REGION Network 15: Oscillator Screen Buttons
   // Set Buttons on based on operations of oscillator
   // Start Button on if Oscillating - State between 200-299
   // Hold Button on if Holding or Bumping - State between 100-199
   // Stop Button on if System Enabled but not Oscillating or Holding/Bumping awaiting Cmd- State 1
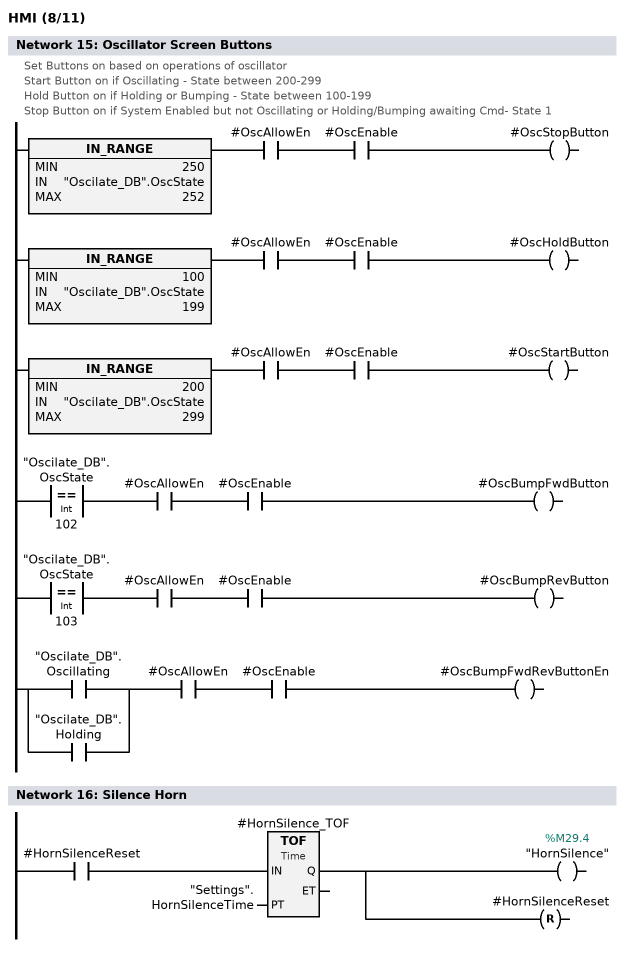
   RUNG wire#powerrail
      { S7_Templates := "SrcType := Int" } InRange(min := 250, in := "Oscilate_DB".OscState, max := 252)
      Contact( #OscAllowEn )
      Contact( #OscEnable )
      Coil( #OscStopButton )
   END_RUNG
   RUNG wire#powerrail
      { S7_Templates := "SrcType := Int" } InRange(min := 100, in := "Oscilate_DB".OscState, max := 199)
      Contact( #OscAllowEn )
      Contact( #OscEnable )
      Coil( #OscHoldButton )
   END_RUNG
   RUNG wire#powerrail
      { S7_Templates := "SrcType := Int" } InRange(min := 200, in := "Oscilate_DB".OscState, max := 299)
      Contact( #OscAllowEn )
      Contact( #OscEnable )
      Coil( #OscStartButton )
   END_RUNG
   RUNG wire#powerrail
      { S7_Templates := "SrcType := Int" } EQ_Contact(in1 := "Oscilate_DB".OscState, in2 := 102)
      Contact( #OscAllowEn )
      Contact( #OscEnable )
      Coil( #OscBumpFwdButton )
   END_RUNG
   RUNG wire#powerrail
      { S7_Templates := "SrcType := Int" } EQ_Contact(in1 := "Oscilate_DB".OscState, in2 := 103)
      Contact( #OscAllowEn )
      Contact( #OscEnable )
      Coil( #OscBumpRevButton )
   END_RUNG
   RUNG wire#powerrail
      Contact( "Oscilate_DB".Oscillating )
      wire#w1
      Contact( #OscAllowEn )
      Contact( #OscEnable )
      Coil( #OscBumpFwdRevButtonEn )
   END_RUNG
   RUNG wire#powerrail
      Contact( "Oscilate_DB".Holding )
   END_RUNG wire#w1
   // the same network as SCL:
   #OscStopButton := (250 <= "Oscilate_DB".OscState) AND ("Oscilate_DB".OscState <= 252) AND #OscAllowEn AND #OscEnable;
   #OscHoldButton := (100 <= "Oscilate_DB".OscState) AND ("Oscilate_DB".OscState <= 199) AND #OscAllowEn AND #OscEnable;
   #OscStartButton := (200 <= "Oscilate_DB".OscState) AND ("Oscilate_DB".OscState <= 299) AND #OscAllowEn AND #OscEnable;
   #OscBumpFwdButton := ("Oscilate_DB".OscState = 102) AND #OscAllowEn AND #OscEnable;
   #OscBumpRevButton := ("Oscilate_DB".OscState = 103) AND #OscAllowEn AND #OscEnable;
   #OscBumpFwdRevButtonEn := ("Oscilate_DB".Oscillating OR "Oscilate_DB".Holding) AND #OscAllowEn AND #OscEnable;
END_REGION

REGION Network 16: Silence Horn
   RUNG wire#powerrail
      Contact( #HornSilenceReset )
      { S7_Templates := "time_type := Time" } #HornSilence_TOF.TOF(pt := "Settings".HornSilenceTime, et =>)
      wire#w1
      Coil( "HornSilence" )
   END_RUNG
   RUNG wire#w1
      R_Coil( #HornSilenceReset )
   END_RUNG
   // the same network as SCL:
   #HornSilence_TOF(IN := #HornSilenceReset, PT := "Settings".HornSilenceTime);   // TOF
   "HornSilence" := #HornSilence_TOF.Q;
   IF #HornSilence_TOF.Q THEN #HornSilenceReset := FALSE; END_IF;
END_REGION

REGION Network 17: Assign Alarms to Alarms1 Int
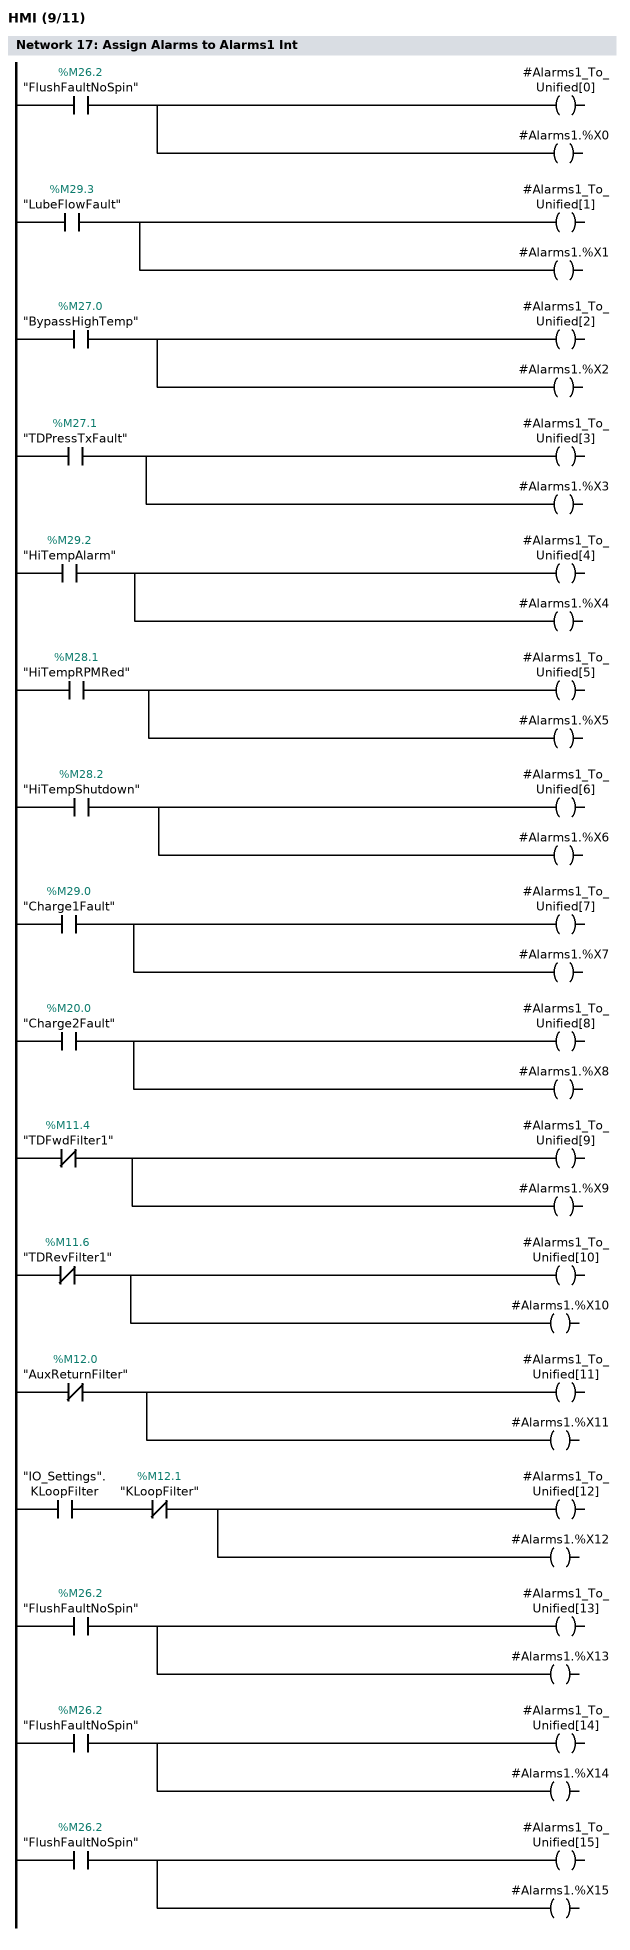
   RUNG wire#powerrail
      Contact( "FlushFaultNoSpin" )
      wire#w1
      Coil( #Alarms1_To_Unified[0] )
   END_RUNG
   RUNG wire#w1
      Coil( #Alarms1.%X0 )
   END_RUNG
   RUNG wire#powerrail
      Contact( "LubeFlowFault" )
      wire#w2
      Coil( #Alarms1_To_Unified[1] )
   END_RUNG
   RUNG wire#w2
      Coil( #Alarms1.%X1 )
   END_RUNG
   RUNG wire#powerrail
      Contact( "BypassHighTemp" )
      wire#w3
      Coil( #Alarms1_To_Unified[2] )
   END_RUNG
   RUNG wire#w3
      Coil( #Alarms1.%X2 )
   END_RUNG
   RUNG wire#powerrail
      Contact( "TDPressTxFault" )
      wire#w4
      Coil( #Alarms1_To_Unified[3] )
   END_RUNG
   RUNG wire#w4
      Coil( #Alarms1.%X3 )
   END_RUNG
   RUNG wire#powerrail
      Contact( "HiTempAlarm" )
      wire#w5
      Coil( #Alarms1_To_Unified[4] )
   END_RUNG
   RUNG wire#w5
      Coil( #Alarms1.%X4 )
   END_RUNG
   RUNG wire#powerrail
      Contact( "HiTempRPMRed" )
      wire#w6
      Coil( #Alarms1_To_Unified[5] )
   END_RUNG
   RUNG wire#w6
      Coil( #Alarms1.%X5 )
   END_RUNG
   RUNG wire#powerrail
      Contact( "HiTempShutdown" )
      wire#w7
      Coil( #Alarms1_To_Unified[6] )
   END_RUNG
   RUNG wire#w7
      Coil( #Alarms1.%X6 )
   END_RUNG
   RUNG wire#powerrail
      Contact( "Charge1Fault" )
      wire#w8
      Coil( #Alarms1_To_Unified[7] )
   END_RUNG
   RUNG wire#w8
      Coil( #Alarms1.%X7 )
   END_RUNG
   RUNG wire#powerrail
      Contact( "Charge2Fault" )
      wire#w9
      Coil( #Alarms1_To_Unified[8] )
   END_RUNG
   RUNG wire#w9
      Coil( #Alarms1.%X8 )
   END_RUNG
   RUNG wire#powerrail
      I_Contact( "TDFwdFilter1" )
      wire#w10
      Coil( #Alarms1_To_Unified[9] )
   END_RUNG
   RUNG wire#w10
      Coil( #Alarms1.%X9 )
   END_RUNG
   RUNG wire#powerrail
      I_Contact( "TDRevFilter1" )
      wire#w11
      Coil( #Alarms1_To_Unified[10] )
   END_RUNG
   RUNG wire#w11
      Coil( #Alarms1.%X10 )
   END_RUNG
   RUNG wire#powerrail
      I_Contact( "AuxReturnFilter" )
      wire#w12
      Coil( #Alarms1_To_Unified[11] )
   END_RUNG
   RUNG wire#w12
      Coil( #Alarms1.%X11 )
   END_RUNG
   RUNG wire#powerrail
      Contact( "IO_Settings".KLoopFilter )
      I_Contact( "KLoopFilter" )
      wire#w13
      Coil( #Alarms1_To_Unified[12] )
   END_RUNG
   RUNG wire#w13
      Coil( #Alarms1.%X12 )
   END_RUNG
   RUNG wire#powerrail
      Contact( "FlushFaultNoSpin" )
      wire#w14
      Coil( #Alarms1_To_Unified[13] )
   END_RUNG
   RUNG wire#w14
      Coil( #Alarms1.%X13 )
   END_RUNG
   RUNG wire#powerrail
      Contact( "FlushFaultNoSpin" )
      wire#w15
      Coil( #Alarms1_To_Unified[14] )
   END_RUNG
   RUNG wire#w15
      Coil( #Alarms1.%X14 )
   END_RUNG
   RUNG wire#powerrail
      Contact( "FlushFaultNoSpin" )
      wire#w16
      Coil( #Alarms1_To_Unified[15] )
   END_RUNG
   RUNG wire#w16
      Coil( #Alarms1.%X15 )
   END_RUNG
   // the same network as SCL:
   #Alarms1_To_Unified[0] := "FlushFaultNoSpin";
   #Alarms1.%X0 := "FlushFaultNoSpin";
   #Alarms1_To_Unified[1] := "LubeFlowFault";
   #Alarms1.%X1 := "LubeFlowFault";
   #Alarms1_To_Unified[2] := "BypassHighTemp";
   #Alarms1.%X2 := "BypassHighTemp";
   #Alarms1_To_Unified[3] := "TDPressTxFault";
   #Alarms1.%X3 := "TDPressTxFault";
   #Alarms1_To_Unified[4] := "HiTempAlarm";
   #Alarms1.%X4 := "HiTempAlarm";
   #Alarms1_To_Unified[5] := "HiTempRPMRed";
   #Alarms1.%X5 := "HiTempRPMRed";
   #Alarms1_To_Unified[6] := "HiTempShutdown";
   #Alarms1.%X6 := "HiTempShutdown";
   #Alarms1_To_Unified[7] := "Charge1Fault";
   #Alarms1.%X7 := "Charge1Fault";
   #Alarms1_To_Unified[8] := "Charge2Fault";
   #Alarms1.%X8 := "Charge2Fault";
   #Alarms1_To_Unified[9] := NOT "TDFwdFilter1";
   #Alarms1.%X9 := NOT "TDFwdFilter1";
   #Alarms1_To_Unified[10] := NOT "TDRevFilter1";
   #Alarms1.%X10 := NOT "TDRevFilter1";
   #Alarms1_To_Unified[11] := NOT "AuxReturnFilter";
   #Alarms1.%X11 := NOT "AuxReturnFilter";
   #Alarms1_To_Unified[12] := "IO_Settings".KLoopFilter AND NOT "KLoopFilter";
   #Alarms1.%X12 := "IO_Settings".KLoopFilter AND NOT "KLoopFilter";
   #Alarms1_To_Unified[13] := "FlushFaultNoSpin";
   #Alarms1.%X13 := "FlushFaultNoSpin";
   #Alarms1_To_Unified[14] := "FlushFaultNoSpin";
   #Alarms1.%X14 := "FlushFaultNoSpin";
   #Alarms1_To_Unified[15] := "FlushFaultNoSpin";
   #Alarms1.%X15 := "FlushFaultNoSpin";
END_REGION

REGION Network 18: Assign Alarms to Alarms2 Int
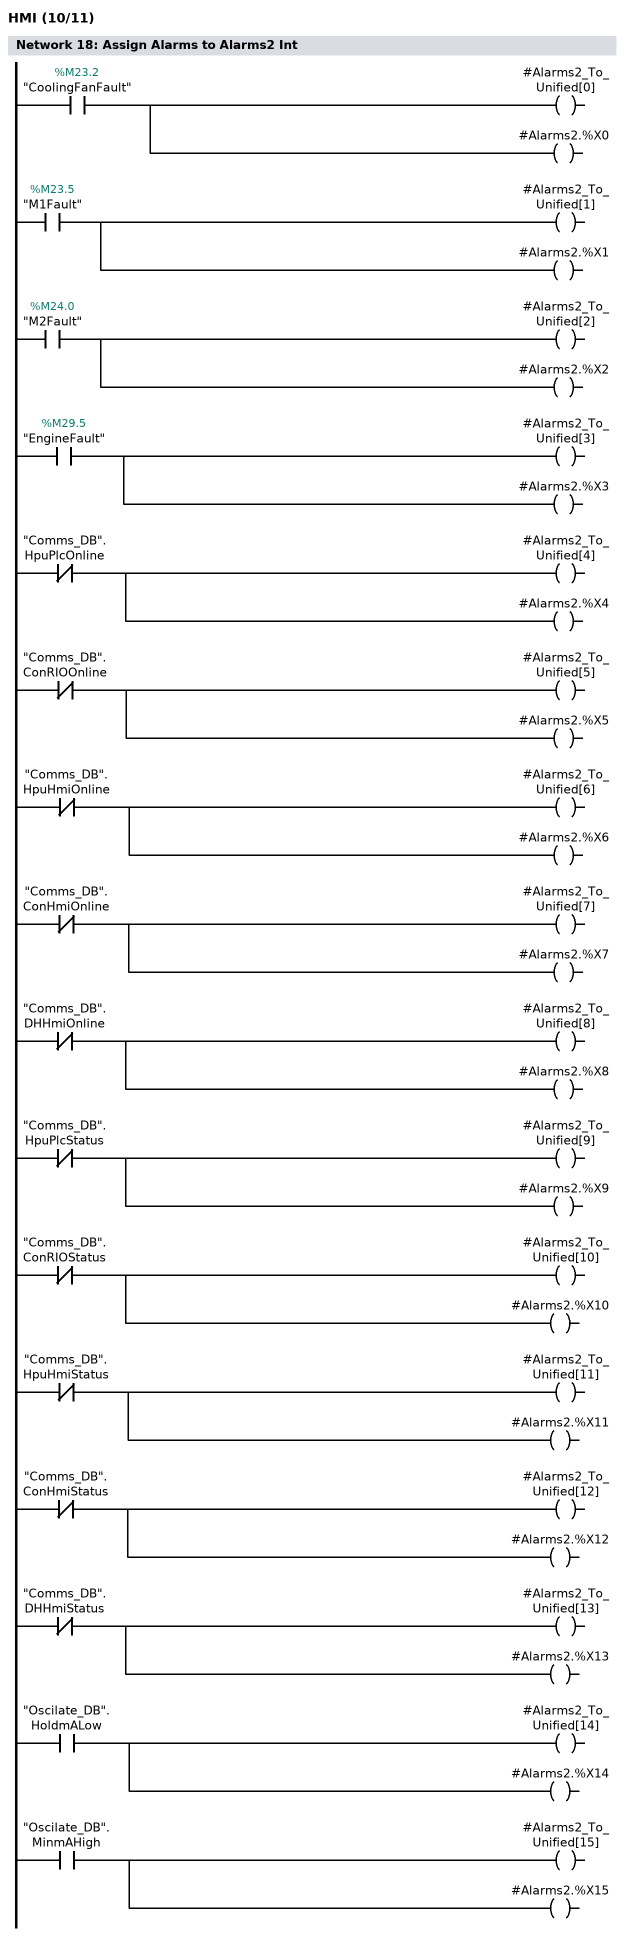
   RUNG wire#powerrail
      Contact( "CoolingFanFault" )
      wire#w1
      Coil( #Alarms2_To_Unified[0] )
   END_RUNG
   RUNG wire#w1
      Coil( #Alarms2.%X0 )
   END_RUNG
   RUNG wire#powerrail
      Contact( "M1Fault" )
      wire#w2
      Coil( #Alarms2_To_Unified[1] )
   END_RUNG
   RUNG wire#w2
      Coil( #Alarms2.%X1 )
   END_RUNG
   RUNG wire#powerrail
      Contact( "M2Fault" )
      wire#w3
      Coil( #Alarms2_To_Unified[2] )
   END_RUNG
   RUNG wire#w3
      Coil( #Alarms2.%X2 )
   END_RUNG
   RUNG wire#powerrail
      Contact( "EngineFault" )
      wire#w4
      Coil( #Alarms2_To_Unified[3] )
   END_RUNG
   RUNG wire#w4
      Coil( #Alarms2.%X3 )
   END_RUNG
   RUNG wire#powerrail
      I_Contact( "Comms_DB".HpuPlcOnline )
      wire#w5
      Coil( #Alarms2_To_Unified[4] )
   END_RUNG
   RUNG wire#w5
      Coil( #Alarms2.%X4 )
   END_RUNG
   RUNG wire#powerrail
      I_Contact( "Comms_DB".ConRIOOnline )
      wire#w6
      Coil( #Alarms2_To_Unified[5] )
   END_RUNG
   RUNG wire#w6
      Coil( #Alarms2.%X5 )
   END_RUNG
   RUNG wire#powerrail
      I_Contact( "Comms_DB".HpuHmiOnline )
      wire#w7
      Coil( #Alarms2_To_Unified[6] )
   END_RUNG
   RUNG wire#w7
      Coil( #Alarms2.%X6 )
   END_RUNG
   RUNG wire#powerrail
      I_Contact( "Comms_DB".ConHmiOnline )
      wire#w8
      Coil( #Alarms2_To_Unified[7] )
   END_RUNG
   RUNG wire#w8
      Coil( #Alarms2.%X7 )
   END_RUNG
   RUNG wire#powerrail
      I_Contact( "Comms_DB".DHHmiOnline )
      wire#w9
      Coil( #Alarms2_To_Unified[8] )
   END_RUNG
   RUNG wire#w9
      Coil( #Alarms2.%X8 )
   END_RUNG
   RUNG wire#powerrail
      I_Contact( "Comms_DB".HpuPlcStatus )
      wire#w10
      Coil( #Alarms2_To_Unified[9] )
   END_RUNG
   RUNG wire#w10
      Coil( #Alarms2.%X9 )
   END_RUNG
   RUNG wire#powerrail
      I_Contact( "Comms_DB".ConRIOStatus )
      wire#w11
      Coil( #Alarms2_To_Unified[10] )
   END_RUNG
   RUNG wire#w11
      Coil( #Alarms2.%X10 )
   END_RUNG
   RUNG wire#powerrail
      I_Contact( "Comms_DB".HpuHmiStatus )
      wire#w12
      Coil( #Alarms2_To_Unified[11] )
   END_RUNG
   RUNG wire#w12
      Coil( #Alarms2.%X11 )
   END_RUNG
   RUNG wire#powerrail
      I_Contact( "Comms_DB".ConHmiStatus )
      wire#w13
      Coil( #Alarms2_To_Unified[12] )
   END_RUNG
   RUNG wire#w13
      Coil( #Alarms2.%X12 )
   END_RUNG
   RUNG wire#powerrail
      I_Contact( "Comms_DB".DHHmiStatus )
      wire#w14
      Coil( #Alarms2_To_Unified[13] )
   END_RUNG
   RUNG wire#w14
      Coil( #Alarms2.%X13 )
   END_RUNG
   RUNG wire#powerrail
      Contact( "Oscilate_DB".HoldmALow )
      wire#w15
      Coil( #Alarms2_To_Unified[14] )
   END_RUNG
   RUNG wire#w15
      Coil( #Alarms2.%X14 )
   END_RUNG
   RUNG wire#powerrail
      Contact( "Oscilate_DB".MinmAHigh )
      wire#w16
      Coil( #Alarms2_To_Unified[15] )
   END_RUNG
   RUNG wire#w16
      Coil( #Alarms2.%X15 )
   END_RUNG
   // the same network as SCL:
   #Alarms2_To_Unified[0] := "CoolingFanFault";
   #Alarms2.%X0 := "CoolingFanFault";
   #Alarms2_To_Unified[1] := "M1Fault";
   #Alarms2.%X1 := "M1Fault";
   #Alarms2_To_Unified[2] := "M2Fault";
   #Alarms2.%X2 := "M2Fault";
   #Alarms2_To_Unified[3] := "EngineFault";
   #Alarms2.%X3 := "EngineFault";
   #Alarms2_To_Unified[4] := NOT "Comms_DB".HpuPlcOnline;
   #Alarms2.%X4 := NOT "Comms_DB".HpuPlcOnline;
   #Alarms2_To_Unified[5] := NOT "Comms_DB".ConRIOOnline;
   #Alarms2.%X5 := NOT "Comms_DB".ConRIOOnline;
   #Alarms2_To_Unified[6] := NOT "Comms_DB".HpuHmiOnline;
   #Alarms2.%X6 := NOT "Comms_DB".HpuHmiOnline;
   #Alarms2_To_Unified[7] := NOT "Comms_DB".ConHmiOnline;
   #Alarms2.%X7 := NOT "Comms_DB".ConHmiOnline;
   #Alarms2_To_Unified[8] := NOT "Comms_DB".DHHmiOnline;
   #Alarms2.%X8 := NOT "Comms_DB".DHHmiOnline;
   #Alarms2_To_Unified[9] := NOT "Comms_DB".HpuPlcStatus;
   #Alarms2.%X9 := NOT "Comms_DB".HpuPlcStatus;
   #Alarms2_To_Unified[10] := NOT "Comms_DB".ConRIOStatus;
   #Alarms2.%X10 := NOT "Comms_DB".ConRIOStatus;
   #Alarms2_To_Unified[11] := NOT "Comms_DB".HpuHmiStatus;
   #Alarms2.%X11 := NOT "Comms_DB".HpuHmiStatus;
   #Alarms2_To_Unified[12] := NOT "Comms_DB".ConHmiStatus;
   #Alarms2.%X12 := NOT "Comms_DB".ConHmiStatus;
   #Alarms2_To_Unified[13] := NOT "Comms_DB".DHHmiStatus;
   #Alarms2.%X13 := NOT "Comms_DB".DHHmiStatus;
   #Alarms2_To_Unified[14] := "Oscilate_DB".HoldmALow;
   #Alarms2.%X14 := "Oscilate_DB".HoldmALow;
   #Alarms2_To_Unified[15] := "Oscilate_DB".MinmAHigh;
   #Alarms2.%X15 := "Oscilate_DB".MinmAHigh;
END_REGION

REGION Network 19: Assign Warnings to Warnings Int
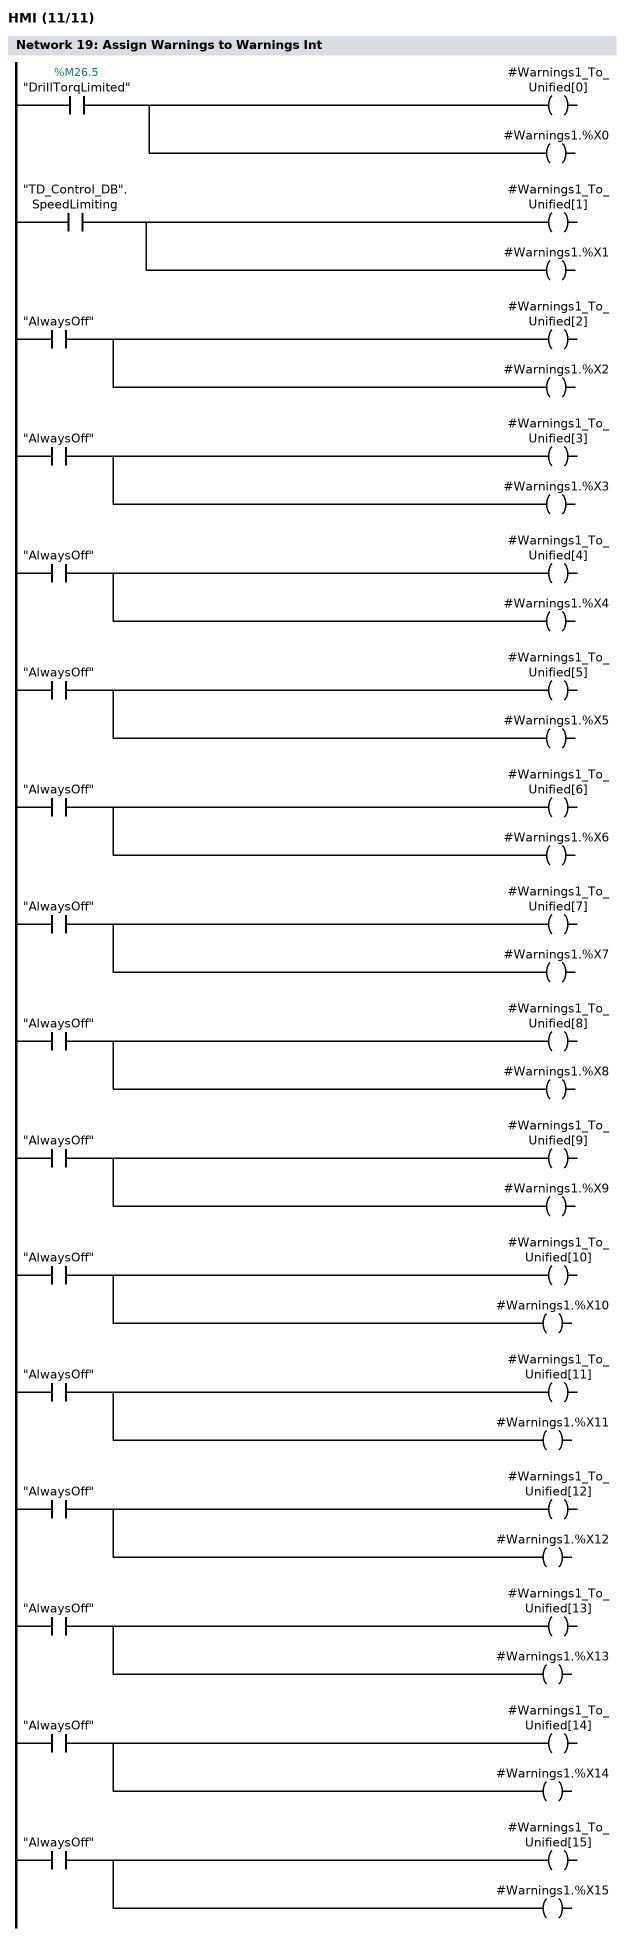
   RUNG wire#powerrail
      Contact( "DrillTorqLimited" )
      wire#w1
      Coil( #Warnings1_To_Unified[0] )
   END_RUNG
   RUNG wire#w1
      Coil( #Warnings1.%X0 )
   END_RUNG
   RUNG wire#powerrail
      Contact( "TD_Control_DB".SpeedLimiting )
      wire#w2
      Coil( #Warnings1_To_Unified[1] )
   END_RUNG
   RUNG wire#w2
      Coil( #Warnings1.%X1 )
   END_RUNG
   RUNG wire#powerrail
      Contact( "AlwaysOff" )
      wire#w3
      Coil( #Warnings1_To_Unified[2] )
   END_RUNG
   RUNG wire#w3
      Coil( #Warnings1.%X2 )
   END_RUNG
   RUNG wire#powerrail
      Contact( "AlwaysOff" )
      wire#w4
      Coil( #Warnings1_To_Unified[3] )
   END_RUNG
   RUNG wire#w4
      Coil( #Warnings1.%X3 )
   END_RUNG
   RUNG wire#powerrail
      Contact( "AlwaysOff" )
      wire#w5
      Coil( #Warnings1_To_Unified[4] )
   END_RUNG
   RUNG wire#w5
      Coil( #Warnings1.%X4 )
   END_RUNG
   RUNG wire#powerrail
      Contact( "AlwaysOff" )
      wire#w6
      Coil( #Warnings1_To_Unified[5] )
   END_RUNG
   RUNG wire#w6
      Coil( #Warnings1.%X5 )
   END_RUNG
   RUNG wire#powerrail
      Contact( "AlwaysOff" )
      wire#w7
      Coil( #Warnings1_To_Unified[6] )
   END_RUNG
   RUNG wire#w7
      Coil( #Warnings1.%X6 )
   END_RUNG
   RUNG wire#powerrail
      Contact( "AlwaysOff" )
      wire#w8
      Coil( #Warnings1_To_Unified[7] )
   END_RUNG
   RUNG wire#w8
      Coil( #Warnings1.%X7 )
   END_RUNG
   RUNG wire#powerrail
      Contact( "AlwaysOff" )
      wire#w9
      Coil( #Warnings1_To_Unified[8] )
   END_RUNG
   RUNG wire#w9
      Coil( #Warnings1.%X8 )
   END_RUNG
   RUNG wire#powerrail
      Contact( "AlwaysOff" )
      wire#w10
      Coil( #Warnings1_To_Unified[9] )
   END_RUNG
   RUNG wire#w10
      Coil( #Warnings1.%X9 )
   END_RUNG
   RUNG wire#powerrail
      Contact( "AlwaysOff" )
      wire#w11
      Coil( #Warnings1_To_Unified[10] )
   END_RUNG
   RUNG wire#w11
      Coil( #Warnings1.%X10 )
   END_RUNG
   RUNG wire#powerrail
      Contact( "AlwaysOff" )
      wire#w12
      Coil( #Warnings1_To_Unified[11] )
   END_RUNG
   RUNG wire#w12
      Coil( #Warnings1.%X11 )
   END_RUNG
   RUNG wire#powerrail
      Contact( "AlwaysOff" )
      wire#w13
      Coil( #Warnings1_To_Unified[12] )
   END_RUNG
   RUNG wire#w13
      Coil( #Warnings1.%X12 )
   END_RUNG
   RUNG wire#powerrail
      Contact( "AlwaysOff" )
      wire#w14
      Coil( #Warnings1_To_Unified[13] )
   END_RUNG
   RUNG wire#w14
      Coil( #Warnings1.%X13 )
   END_RUNG
   RUNG wire#powerrail
      Contact( "AlwaysOff" )
      wire#w15
      Coil( #Warnings1_To_Unified[14] )
   END_RUNG
   RUNG wire#w15
      Coil( #Warnings1.%X14 )
   END_RUNG
   RUNG wire#powerrail
      Contact( "AlwaysOff" )
      wire#w16
      Coil( #Warnings1_To_Unified[15] )
   END_RUNG
   RUNG wire#w16
      Coil( #Warnings1.%X15 )
   END_RUNG
   // the same network as SCL:
   #Warnings1_To_Unified[0] := "DrillTorqLimited";
   #Warnings1.%X0 := "DrillTorqLimited";
   #Warnings1_To_Unified[1] := "TD_Control_DB".SpeedLimiting;
   #Warnings1.%X1 := "TD_Control_DB".SpeedLimiting;
   #Warnings1_To_Unified[2] := "AlwaysOff";
   #Warnings1.%X2 := "AlwaysOff";
   #Warnings1_To_Unified[3] := "AlwaysOff";
   #Warnings1.%X3 := "AlwaysOff";
   #Warnings1_To_Unified[4] := "AlwaysOff";
   #Warnings1.%X4 := "AlwaysOff";
   #Warnings1_To_Unified[5] := "AlwaysOff";
   #Warnings1.%X5 := "AlwaysOff";
   #Warnings1_To_Unified[6] := "AlwaysOff";
   #Warnings1.%X6 := "AlwaysOff";
   #Warnings1_To_Unified[7] := "AlwaysOff";
   #Warnings1.%X7 := "AlwaysOff";
   #Warnings1_To_Unified[8] := "AlwaysOff";
   #Warnings1.%X8 := "AlwaysOff";
   #Warnings1_To_Unified[9] := "AlwaysOff";
   #Warnings1.%X9 := "AlwaysOff";
   #Warnings1_To_Unified[10] := "AlwaysOff";
   #Warnings1.%X10 := "AlwaysOff";
   #Warnings1_To_Unified[11] := "AlwaysOff";
   #Warnings1.%X11 := "AlwaysOff";
   #Warnings1_To_Unified[12] := "AlwaysOff";
   #Warnings1.%X12 := "AlwaysOff";
   #Warnings1_To_Unified[13] := "AlwaysOff";
   #Warnings1.%X13 := "AlwaysOff";
   #Warnings1_To_Unified[14] := "AlwaysOff";
   #Warnings1.%X14 := "AlwaysOff";
   #Warnings1_To_Unified[15] := "AlwaysOff";
   #Warnings1.%X15 := "AlwaysOff";
END_REGION
END_FUNCTION_BLOCK

FUNCTION_BLOCK "Calculations"   // FB10, LAD
{ S7_Optimized_Access := 'TRUE' }
// stored: AutoNumber false, MemoryReserve 100, SetENOAutomatically false
   VAR
      M1_LPF { S7_SetPoint := 'True'} : "LowPassFilter";
      M2_LPF { S7_SetPoint := 'True'} : "LowPassFilter";
      TDPressFwd_LPF { S7_SetPoint := 'True'} : "LowPassFilter";
      TDPressRev_LPF { S7_SetPoint := 'True'} : "LowPassFilter";
      ClosedLoopTemp_LPF { S7_SetPoint := 'True'} : "LowPassFilter";
      ChargeFlow_LPF { S7_SetPoint := 'True'} : "LowPassFilter";
      HotOilFlow_LPF { S7_SetPoint := 'True'} : "LowPassFilter";
      AuxFlow_LPF { S7_SetPoint := 'True'} : "LowPassFilter";
      ChargePress1_LPF { S7_SetPoint := 'True'} : "LowPassFilter";
      ChargePress2_LPF { S7_SetPoint := 'True'} : "LowPassFilter";
      DrillTorqPotLPF { S7_SetPoint := 'True'} : "LowPassFilter";
      MUTorqPotLPF { S7_SetPoint := 'True'} : "LowPassFilter";
      DrillThrottlePotLPF { S7_SetPoint := 'True'} : "LowPassFilter";
      ActTorq_LPF { S7_SetPoint := 'True'} : "LowPassFilter";
      DrillRecPTO_TP { S7_SetPoint := 'True'} : TP_TIME;
      DrillRecMax { S7_SetPoint := 'True'} : Bool;   // Send max value out to drill recorder
   END_VAR
   VAR_TEMP
      tempReal : Real;
      AutoMUTorqSetLow : Real;
      AutoMUTorqSetHigh : Real;
   END_VAR
   VAR_TEMP   // added for the SCL form of the ladder/FBD networks
      _w1 : Bool;
      _w2 : Bool;
      _w3 : Bool;
      _w4 : Bool;
      _w5 : Bool;
      _w6 : Bool;
   END_VAR
BEGIN

REGION Network 1: Encoder Position
   // Hard coded rollover value to match encoder rollver value from TM Count card
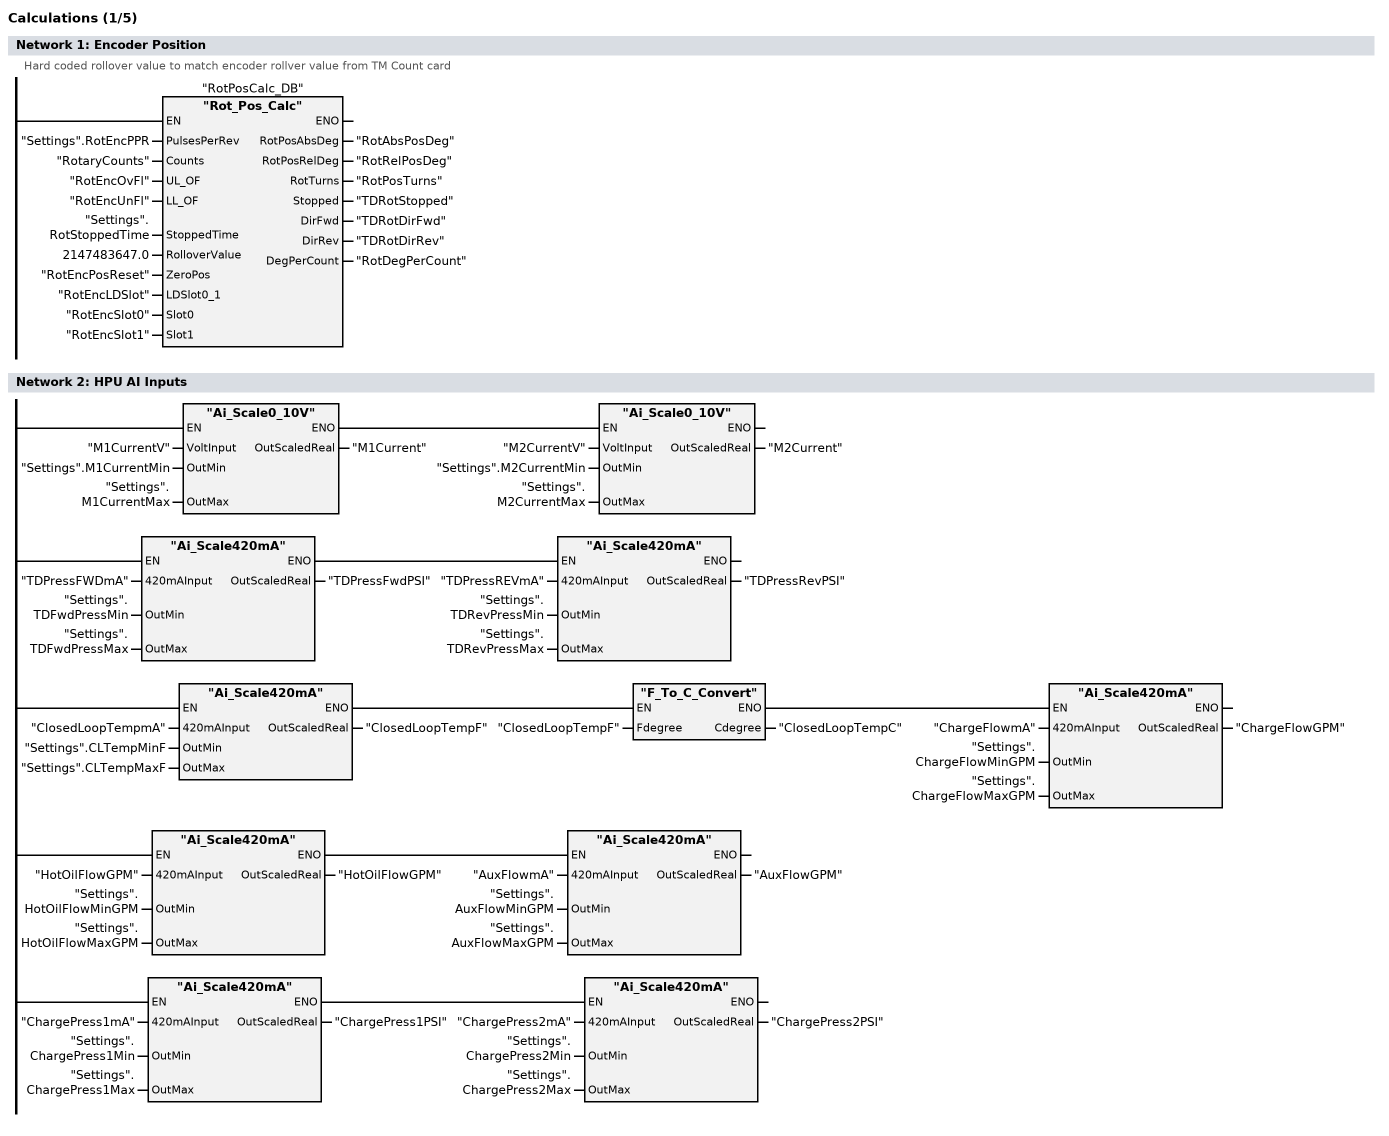
   RUNG wire#powerrail
      "RotPosCalc_DB"(PulsesPerRev := "Settings".RotEncPPR, Counts := "RotaryCounts", UL_OF := "RotEncOvFl", LL_OF := "RotEncUnFl", StoppedTime := "Settings".RotStoppedTime, RolloverValue := 2147483647.0, ZeroPos := "RotEncPosReset", LDSlot0_1 := "RotEncLDSlot", Slot0 := "RotEncSlot0", Slot1 := "RotEncSlot1", RotPosAbsDeg => "RotAbsPosDeg", RotPosRelDeg => "RotRelPosDeg", RotTurns => "RotPosTurns", Stopped => "TDRotStopped", DirFwd => "TDRotDirFwd", DirRev => "TDRotDirRev", DegPerCount => "RotDegPerCount")
   END_RUNG
   // the same network as SCL:
   "RotPosCalc_DB"(PulsesPerRev := "Settings".RotEncPPR,   // "Rot_Pos_Calc"
                   Counts := "RotaryCounts",
                   UL_OF := "RotEncOvFl",
                   LL_OF := "RotEncUnFl",
                   StoppedTime := "Settings".RotStoppedTime,
                   RolloverValue := 2147483647.0,
                   ZeroPos := "RotEncPosReset",
                   LDSlot0_1 := "RotEncLDSlot",
                   Slot0 := "RotEncSlot0",
                   Slot1 := "RotEncSlot1",
                   RotPosAbsDeg => "RotAbsPosDeg",
                   RotPosRelDeg => "RotRelPosDeg",
                   RotTurns => "RotPosTurns",
                   Stopped => "TDRotStopped",
                   DirFwd => "TDRotDirFwd",
                   DirRev => "TDRotDirRev",
                   DegPerCount => "RotDegPerCount");
END_REGION

REGION Network 2: HPU AI Inputs
   RUNG wire#powerrail
      "Ai_Scale0_10V"(VoltInput := "M1CurrentV", OutMin := "Settings".M1CurrentMin, OutMax := "Settings".M1CurrentMax, OutScaledReal => "M1Current")
      "Ai_Scale0_10V"(VoltInput := "M2CurrentV", OutMin := "Settings".M2CurrentMin, OutMax := "Settings".M2CurrentMax, OutScaledReal => "M2Current")
   END_RUNG
   RUNG wire#powerrail
      "Ai_Scale420mA"("420mAInput" := "TDPressFWDmA", OutMin := "Settings".TDFwdPressMin, OutMax := "Settings".TDFwdPressMax, OutScaledReal => "TDPressFwdPSI")
      "Ai_Scale420mA"("420mAInput" := "TDPressREVmA", OutMin := "Settings".TDRevPressMin, OutMax := "Settings".TDRevPressMax, OutScaledReal => "TDPressRevPSI")
   END_RUNG
   RUNG wire#powerrail
      "Ai_Scale420mA"("420mAInput" := "ClosedLoopTempmA", OutMin := "Settings".CLTempMinF, OutMax := "Settings".CLTempMaxF, OutScaledReal => "ClosedLoopTempF")
      "F_To_C_Convert"(Fdegree := "ClosedLoopTempF", Cdegree => "ClosedLoopTempC")
      "Ai_Scale420mA"("420mAInput" := "ChargeFlowmA", OutMin := "Settings".ChargeFlowMinGPM, OutMax := "Settings".ChargeFlowMaxGPM, OutScaledReal => "ChargeFlowGPM")
   END_RUNG
   RUNG wire#powerrail
      "Ai_Scale420mA"("420mAInput" := "HotOilFlowGPM", OutMin := "Settings".HotOilFlowMinGPM, OutMax := "Settings".HotOilFlowMaxGPM, OutScaledReal => "HotOilFlowGPM")
      "Ai_Scale420mA"("420mAInput" := "AuxFlowmA", OutMin := "Settings".AuxFlowMinGPM, OutMax := "Settings".AuxFlowMaxGPM, OutScaledReal => "AuxFlowGPM")
   END_RUNG
   RUNG wire#powerrail
      "Ai_Scale420mA"("420mAInput" := "ChargePress1mA", OutMin := "Settings".ChargePress1Min, OutMax := "Settings".ChargePress1Max, OutScaledReal => "ChargePress1PSI")
      "Ai_Scale420mA"("420mAInput" := "ChargePress2mA", OutMin := "Settings".ChargePress2Min, OutMax := "Settings".ChargePress2Max, OutScaledReal => "ChargePress2PSI")
   END_RUNG
   // the same network as SCL:
   "Ai_Scale0_10V"(VoltInput := "M1CurrentV",
                   OutMin := "Settings".M1CurrentMin,
                   OutMax := "Settings".M1CurrentMax,
                   OutScaledReal => "M1Current",
                   ENO => #_w1);
   IF #_w1 THEN
       "Ai_Scale0_10V"(VoltInput := "M2CurrentV",
                       OutMin := "Settings".M2CurrentMin,
                       OutMax := "Settings".M2CurrentMax,
                       OutScaledReal => "M2Current");
   END_IF;
   "Ai_Scale420mA"("420mAInput" := "TDPressFWDmA",
                   OutMin := "Settings".TDFwdPressMin,
                   OutMax := "Settings".TDFwdPressMax,
                   OutScaledReal => "TDPressFwdPSI",
                   ENO => #_w2);
   IF #_w2 THEN
       "Ai_Scale420mA"("420mAInput" := "TDPressREVmA",
                       OutMin := "Settings".TDRevPressMin,
                       OutMax := "Settings".TDRevPressMax,
                       OutScaledReal => "TDPressRevPSI");
   END_IF;
   "Ai_Scale420mA"("420mAInput" := "ClosedLoopTempmA",
                   OutMin := "Settings".CLTempMinF,
                   OutMax := "Settings".CLTempMaxF,
                   OutScaledReal => "ClosedLoopTempF",
                   ENO => #_w3);
   "F_To_C_Convert"(EN := #_w3, Fdegree := "ClosedLoopTempF", Cdegree => "ClosedLoopTempC", ENO => #_w4);
   IF #_w4 THEN
       "Ai_Scale420mA"("420mAInput" := "ChargeFlowmA",
                       OutMin := "Settings".ChargeFlowMinGPM,
                       OutMax := "Settings".ChargeFlowMaxGPM,
                       OutScaledReal => "ChargeFlowGPM");
   END_IF;
   "Ai_Scale420mA"("420mAInput" := "HotOilFlowGPM",
                   OutMin := "Settings".HotOilFlowMinGPM,
                   OutMax := "Settings".HotOilFlowMaxGPM,
                   OutScaledReal => "HotOilFlowGPM",
                   ENO => #_w5);
   IF #_w5 THEN
       "Ai_Scale420mA"("420mAInput" := "AuxFlowmA",
                       OutMin := "Settings".AuxFlowMinGPM,
                       OutMax := "Settings".AuxFlowMaxGPM,
                       OutScaledReal => "AuxFlowGPM");
   END_IF;
   "Ai_Scale420mA"("420mAInput" := "ChargePress1mA",
                   OutMin := "Settings".ChargePress1Min,
                   OutMax := "Settings".ChargePress1Max,
                   OutScaledReal => "ChargePress1PSI",
                   ENO => #_w6);
   IF #_w6 THEN
       "Ai_Scale420mA"("420mAInput" := "ChargePress2mA",
                       OutMin := "Settings".ChargePress2Min,
                       OutMax := "Settings".ChargePress2Max,
                       OutScaledReal => "ChargePress2PSI");
   END_IF;
END_REGION

REGION Network 3: Filter HPU Inputs
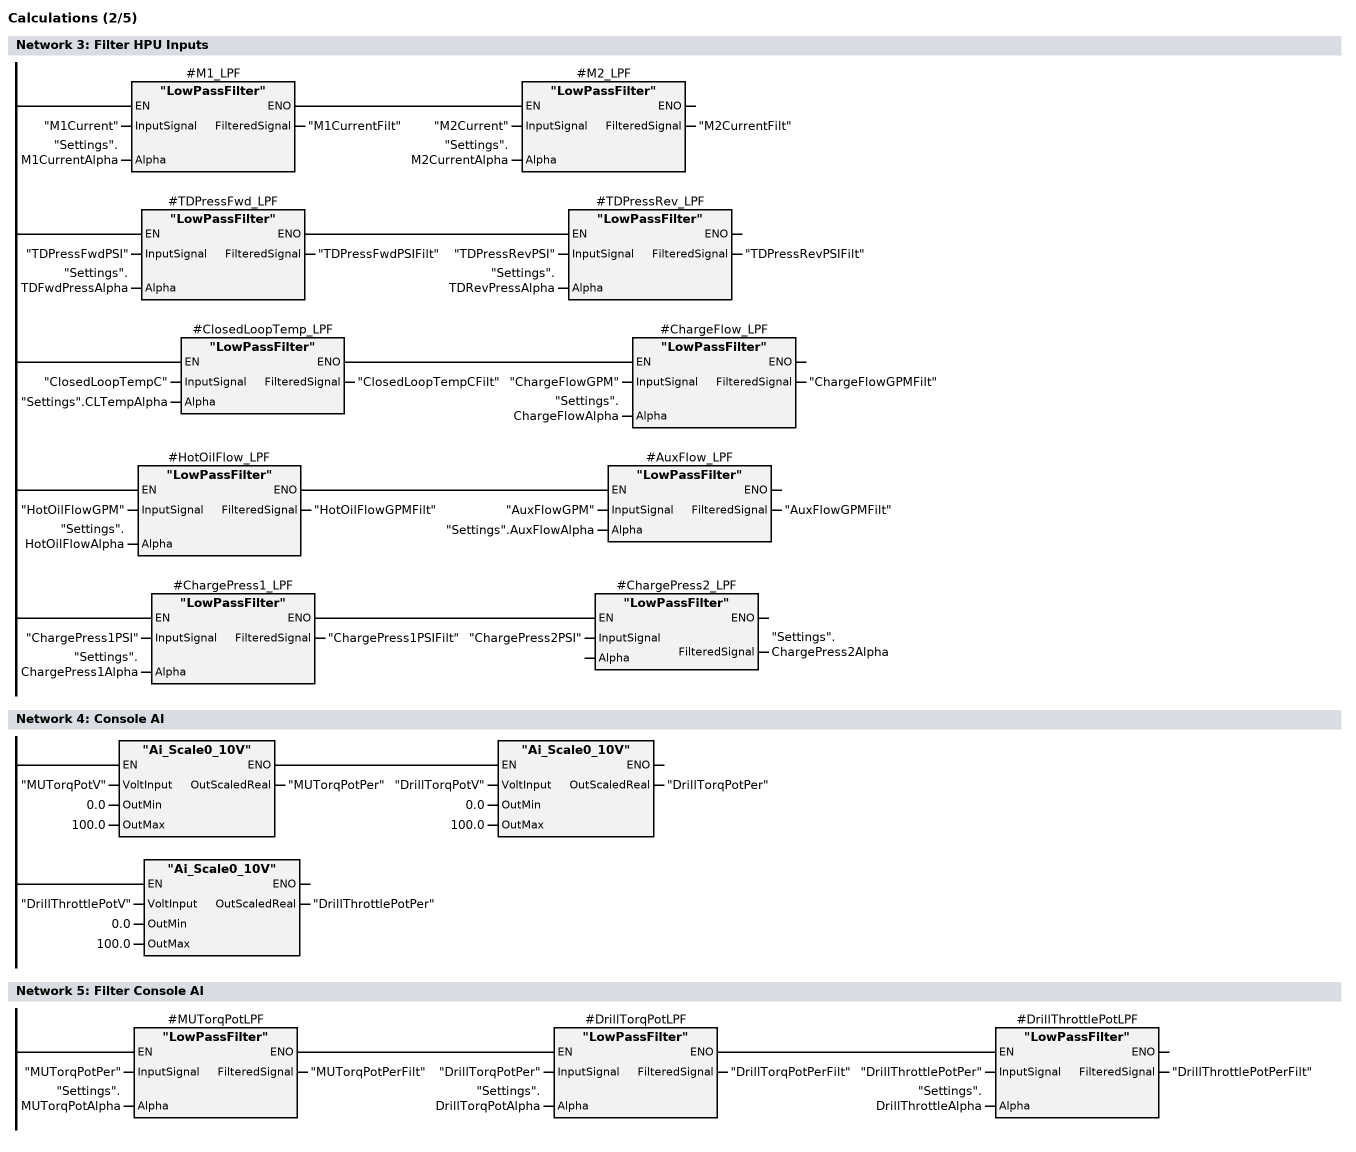
   RUNG wire#powerrail
      #M1_LPF(InputSignal := "M1Current", Alpha := "Settings".M1CurrentAlpha, FilteredSignal => "M1CurrentFilt")
      #M2_LPF(InputSignal := "M2Current", Alpha := "Settings".M2CurrentAlpha, FilteredSignal => "M2CurrentFilt")
   END_RUNG
   RUNG wire#powerrail
      #TDPressFwd_LPF(InputSignal := "TDPressFwdPSI", Alpha := "Settings".TDFwdPressAlpha, FilteredSignal => "TDPressFwdPSIFilt")
      #TDPressRev_LPF(InputSignal := "TDPressRevPSI", Alpha := "Settings".TDRevPressAlpha, FilteredSignal => "TDPressRevPSIFilt")
   END_RUNG
   RUNG wire#powerrail
      #ClosedLoopTemp_LPF(InputSignal := "ClosedLoopTempC", Alpha := "Settings".CLTempAlpha, FilteredSignal => "ClosedLoopTempCFilt")
      #ChargeFlow_LPF(InputSignal := "ChargeFlowGPM", Alpha := "Settings".ChargeFlowAlpha, FilteredSignal => "ChargeFlowGPMFilt")
   END_RUNG
   RUNG wire#powerrail
      #HotOilFlow_LPF(InputSignal := "HotOilFlowGPM", Alpha := "Settings".HotOilFlowAlpha, FilteredSignal => "HotOilFlowGPMFilt")
      #AuxFlow_LPF(InputSignal := "AuxFlowGPM", Alpha := "Settings".AuxFlowAlpha, FilteredSignal => "AuxFlowGPMFilt")
   END_RUNG
   RUNG wire#powerrail
      #ChargePress1_LPF(InputSignal := "ChargePress1PSI", Alpha := "Settings".ChargePress1Alpha, FilteredSignal => "ChargePress1PSIFilt")
      #ChargePress2_LPF(InputSignal := "ChargePress2PSI", Alpha :=, FilteredSignal => "Settings".ChargePress2Alpha)
   END_RUNG
   // the same network as SCL:
   #M1_LPF(InputSignal := "M1Current",   // "LowPassFilter"
           Alpha := "Settings".M1CurrentAlpha,
           FilteredSignal => "M1CurrentFilt",
           ENO => #_w1);
   IF #_w1 THEN
       #M2_LPF(InputSignal := "M2Current", Alpha := "Settings".M2CurrentAlpha, FilteredSignal => "M2CurrentFilt");   // "LowPassFilter"
   END_IF;
   #TDPressFwd_LPF(InputSignal := "TDPressFwdPSI",   // "LowPassFilter"
                   Alpha := "Settings".TDFwdPressAlpha,
                   FilteredSignal => "TDPressFwdPSIFilt",
                   ENO => #_w2);
   IF #_w2 THEN
       #TDPressRev_LPF(InputSignal := "TDPressRevPSI",   // "LowPassFilter"
                       Alpha := "Settings".TDRevPressAlpha,
                       FilteredSignal => "TDPressRevPSIFilt");
   END_IF;
   #ClosedLoopTemp_LPF(InputSignal := "ClosedLoopTempC",   // "LowPassFilter"
                       Alpha := "Settings".CLTempAlpha,
                       FilteredSignal => "ClosedLoopTempCFilt",
                       ENO => #_w3);
   IF #_w3 THEN
       #ChargeFlow_LPF(InputSignal := "ChargeFlowGPM",   // "LowPassFilter"
                       Alpha := "Settings".ChargeFlowAlpha,
                       FilteredSignal => "ChargeFlowGPMFilt");
   END_IF;
   #HotOilFlow_LPF(InputSignal := "HotOilFlowGPM",   // "LowPassFilter"
                   Alpha := "Settings".HotOilFlowAlpha,
                   FilteredSignal => "HotOilFlowGPMFilt",
                   ENO => #_w4);
   IF #_w4 THEN
       #AuxFlow_LPF(InputSignal := "AuxFlowGPM",   // "LowPassFilter"
                    Alpha := "Settings".AuxFlowAlpha,
                    FilteredSignal => "AuxFlowGPMFilt");
   END_IF;
   #ChargePress1_LPF(InputSignal := "ChargePress1PSI",   // "LowPassFilter"
                     Alpha := "Settings".ChargePress1Alpha,
                     FilteredSignal => "ChargePress1PSIFilt",
                     ENO => #_w5);
   IF #_w5 THEN
       #ChargePress2_LPF(InputSignal := "ChargePress2PSI", FilteredSignal => "Settings".ChargePress2Alpha);   // "LowPassFilter"
   END_IF;
END_REGION

REGION Network 4: Console AI
   RUNG wire#powerrail
      "Ai_Scale0_10V"(VoltInput := "MUTorqPotV", OutMin := 0.0, OutMax := 100.0, OutScaledReal => "MUTorqPotPer")
      "Ai_Scale0_10V"(VoltInput := "DrillTorqPotV", OutMin := 0.0, OutMax := 100.0, OutScaledReal => "DrillTorqPotPer")
   END_RUNG
   RUNG wire#powerrail
      "Ai_Scale0_10V"(VoltInput := "DrillThrottlePotV", OutMin := 0.0, OutMax := 100.0, OutScaledReal => "DrillThrottlePotPer")
   END_RUNG
   // the same network as SCL:
   "Ai_Scale0_10V"(VoltInput := "MUTorqPotV",
                   OutMin := 0.0,
                   OutMax := 100.0,
                   OutScaledReal => "MUTorqPotPer",
                   ENO => #_w1);
   IF #_w1 THEN
       "Ai_Scale0_10V"(VoltInput := "DrillTorqPotV",
                       OutMin := 0.0,
                       OutMax := 100.0,
                       OutScaledReal => "DrillTorqPotPer");
   END_IF;
   "Ai_Scale0_10V"(VoltInput := "DrillThrottlePotV",
                   OutMin := 0.0,
                   OutMax := 100.0,
                   OutScaledReal => "DrillThrottlePotPer");
END_REGION

REGION Network 5: Filter Console AI
   RUNG wire#powerrail
      #MUTorqPotLPF(InputSignal := "MUTorqPotPer", Alpha := "Settings".MUTorqPotAlpha, FilteredSignal => "MUTorqPotPerFilt")
      #DrillTorqPotLPF(InputSignal := "DrillTorqPotPer", Alpha := "Settings".DrillTorqPotAlpha, FilteredSignal => "DrillTorqPotPerFilt")
      #DrillThrottlePotLPF(InputSignal := "DrillThrottlePotPer", Alpha := "Settings".DrillThrottleAlpha, FilteredSignal => "DrillThrottlePotPerFilt")
   END_RUNG
   // the same network as SCL:
   #MUTorqPotLPF(InputSignal := "MUTorqPotPer",   // "LowPassFilter"
                 Alpha := "Settings".MUTorqPotAlpha,
                 FilteredSignal => "MUTorqPotPerFilt",
                 ENO => #_w1);
   #DrillTorqPotLPF(EN := #_w1,   // "LowPassFilter"
                    InputSignal := "DrillTorqPotPer",
                    Alpha := "Settings".DrillTorqPotAlpha,
                    FilteredSignal => "DrillTorqPotPerFilt",
                    ENO => #_w2);
   IF #_w2 THEN
       #DrillThrottlePotLPF(InputSignal := "DrillThrottlePotPer",   // "LowPassFilter"
                            Alpha := "Settings".DrillThrottleAlpha,
                            FilteredSignal => "DrillThrottlePotPerFilt");
   END_IF;
END_REGION

REGION Network 6: Torque Calculation
   // Differential Pressure x torque factor(ft-lbs/psi) unless bypass running * efficiency. Use raw reading value and filter after
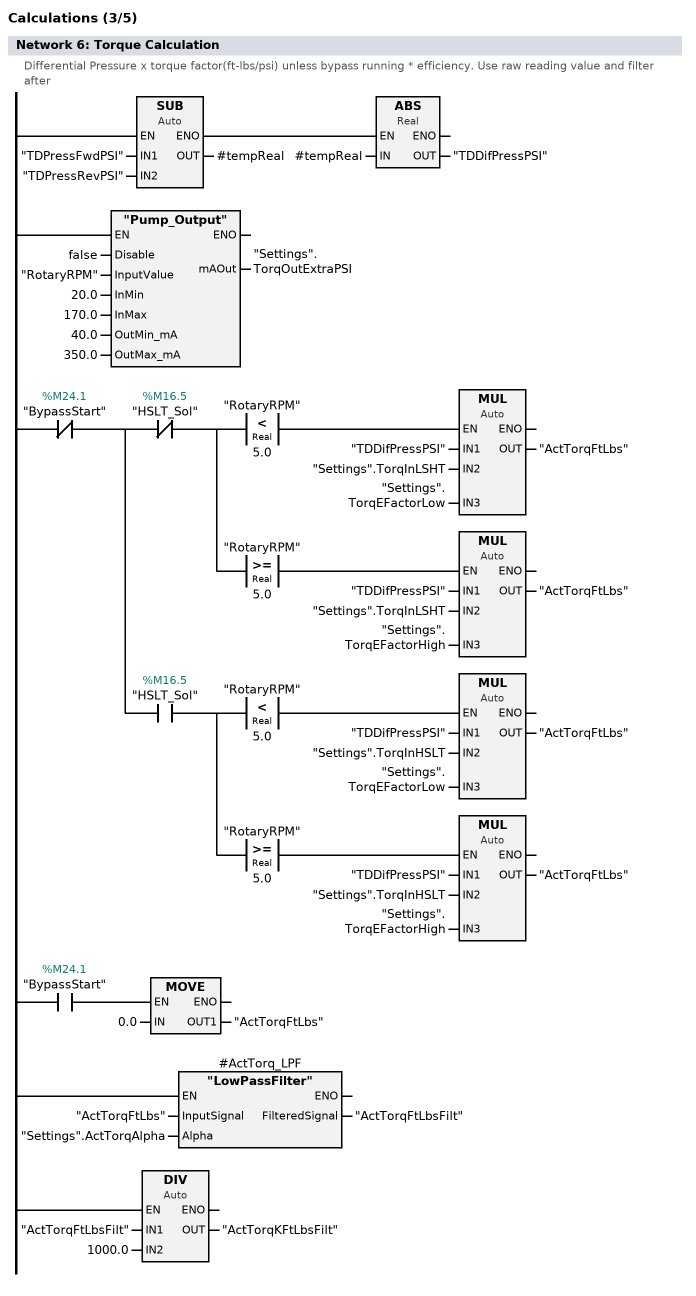
   RUNG wire#powerrail
      Sub(in1 := "TDPressFwdPSI", in2 := "TDPressRevPSI", out => #tempReal)
      { S7_Templates := "SrcType := Real" } Abs(in := #tempReal, out => "TDDifPressPSI")
   END_RUNG
   RUNG wire#powerrail
      "Pump_Output"(Disable := false, InputValue := "RotaryRPM", InMin := 20.0, InMax := 170.0, OutMin_mA := 40.0, OutMax_mA := 350.0, mAOut => "Settings".TorqOutExtraPSI)
   END_RUNG
   RUNG wire#powerrail
      I_Contact( "BypassStart" )
      wire#w1
      I_Contact( "HSLT_Sol" )
      wire#w2
      { S7_Templates := "SrcType := Real" } LT_Contact(in1 := "RotaryRPM", in2 := 5.0)
      Mul(in1 := "TDDifPressPSI", in2 := "Settings".TorqInLSHT, in3 := "Settings".TorqEFactorLow, out => "ActTorqFtLbs")
   END_RUNG
   RUNG wire#w2
      { S7_Templates := "SrcType := Real" } GE_Contact(in1 := "RotaryRPM", in2 := 5.0)
      Mul(in1 := "TDDifPressPSI", in2 := "Settings".TorqInLSHT, in3 := "Settings".TorqEFactorHigh, out => "ActTorqFtLbs")
   END_RUNG
   RUNG wire#w1
      Contact( "HSLT_Sol" )
      wire#w3
      { S7_Templates := "SrcType := Real" } LT_Contact(in1 := "RotaryRPM", in2 := 5.0)
      Mul(in1 := "TDDifPressPSI", in2 := "Settings".TorqInHSLT, in3 := "Settings".TorqEFactorLow, out => "ActTorqFtLbs")
   END_RUNG
   RUNG wire#w3
      { S7_Templates := "SrcType := Real" } GE_Contact(in1 := "RotaryRPM", in2 := 5.0)
      Mul(in1 := "TDDifPressPSI", in2 := "Settings".TorqInHSLT, in3 := "Settings".TorqEFactorHigh, out => "ActTorqFtLbs")
   END_RUNG
   RUNG wire#powerrail
      Contact( "BypassStart" )
      Move(in := 0.0, out1 => "ActTorqFtLbs")
   END_RUNG
   RUNG wire#powerrail
      #ActTorq_LPF(InputSignal := "ActTorqFtLbs", Alpha := "Settings".ActTorqAlpha, FilteredSignal => "ActTorqFtLbsFilt")
   END_RUNG
   RUNG wire#powerrail
      Div(in1 := "ActTorqFtLbsFilt", in2 := 1000.0, out => "ActTorqKFtLbsFilt")
   END_RUNG
   // the same network as SCL:
   #tempReal := "TDPressFwdPSI" - "TDPressRevPSI";
   "TDDifPressPSI" := ABS(#tempReal);
   "Pump_Output"(Disable := false,
                 InputValue := "RotaryRPM",
                 InMin := 20.0,
                 InMax := 170.0,
                 OutMin_mA := 40.0,
                 OutMax_mA := 350.0,
                 mAOut => "Settings".TorqOutExtraPSI);
   #_w1 := NOT "BypassStart" AND NOT "HSLT_Sol";
   IF #_w1 AND ("RotaryRPM" < 5.0) THEN
       "ActTorqFtLbs" := "TDDifPressPSI" * "Settings".TorqInLSHT * "Settings".TorqEFactorLow;
   END_IF;
   IF #_w1 AND ("RotaryRPM" >= 5.0) THEN
       "ActTorqFtLbs" := "TDDifPressPSI" * "Settings".TorqInLSHT * "Settings".TorqEFactorHigh;
   END_IF;
   #_w2 := NOT "BypassStart" AND "HSLT_Sol";
   IF #_w2 AND ("RotaryRPM" < 5.0) THEN
       "ActTorqFtLbs" := "TDDifPressPSI" * "Settings".TorqInHSLT * "Settings".TorqEFactorLow;
   END_IF;
   IF #_w2 AND ("RotaryRPM" >= 5.0) THEN
       "ActTorqFtLbs" := "TDDifPressPSI" * "Settings".TorqInHSLT * "Settings".TorqEFactorHigh;
   END_IF;
   IF "BypassStart" THEN "ActTorqFtLbs" := 0.0; END_IF;
   #ActTorq_LPF(InputSignal := "ActTorqFtLbs",   // "LowPassFilter"
                Alpha := "Settings".ActTorqAlpha,
                FilteredSignal => "ActTorqFtLbsFilt");
   "ActTorqKFtLbsFilt" := "ActTorqFtLbsFilt" / 1000.0;
END_REGION

REGION Network 7: User Setpoints
   // Drill torque setpoint cannot be greater than 0.95 % of the makeup setpoint
   // MU Torque always low speed as it cannot shift
   // Drill torque depends on speed settings
   // MU threshold is a percent of setpoint
   // Add 500 PSI to setpoint to overcome charge pressure
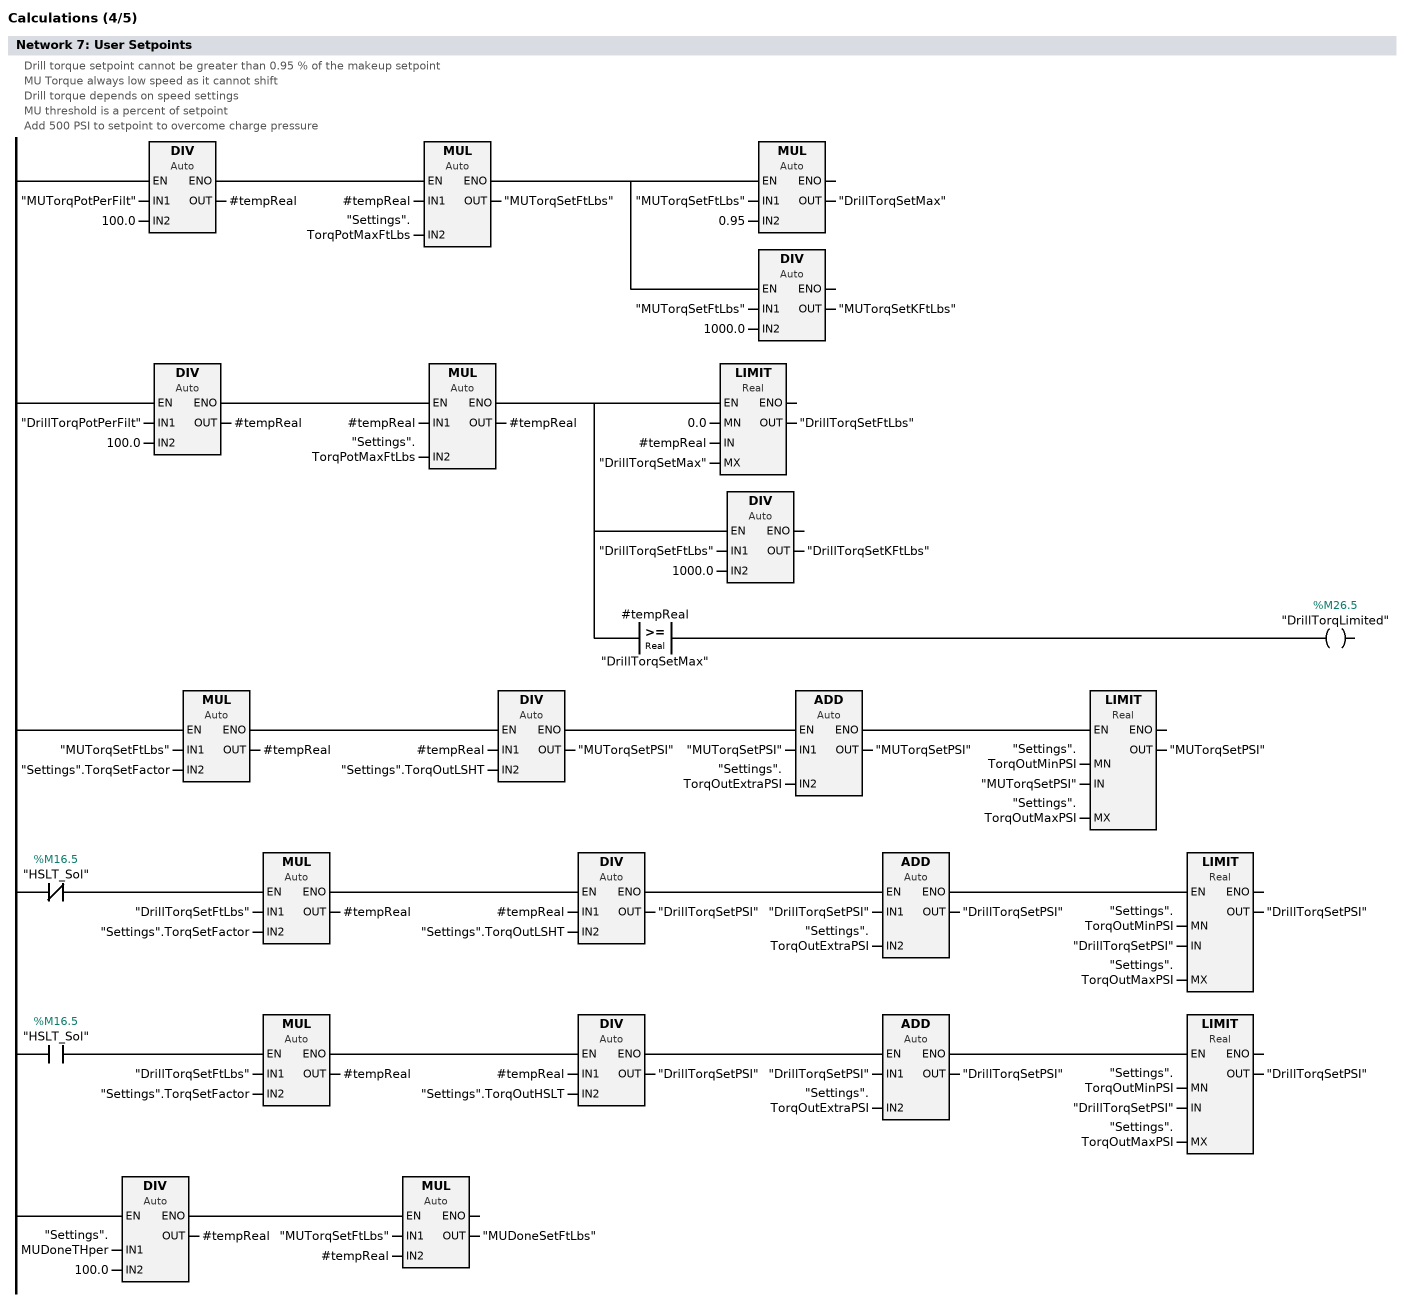
   RUNG wire#powerrail
      Div(in1 := "MUTorqPotPerFilt", in2 := 100.0, out => #tempReal)
      Mul(in1 := #tempReal, in2 := "Settings".TorqPotMaxFtLbs, out => "MUTorqSetFtLbs")
      wire#w1
      Mul(in1 := "MUTorqSetFtLbs", in2 := 0.95, out => "DrillTorqSetMax")
   END_RUNG
   RUNG wire#w1
      Div(in1 := "MUTorqSetFtLbs", in2 := 1000.0, out => "MUTorqSetKFtLbs")
   END_RUNG
   RUNG wire#powerrail
      Div(in1 := "DrillTorqPotPerFilt", in2 := 100.0, out => #tempReal)
      Mul(in1 := #tempReal, in2 := "Settings".TorqPotMaxFtLbs, out => #tempReal)
      wire#w2
      { S7_Templates := "value_type := Real" } Limit(mn := 0.0, in := #tempReal, mx := "DrillTorqSetMax", out => "DrillTorqSetFtLbs")
   END_RUNG
   RUNG wire#w2
      Div(in1 := "DrillTorqSetFtLbs", in2 := 1000.0, out => "DrillTorqSetKFtLbs")
   END_RUNG
   RUNG wire#w2
      { S7_Templates := "SrcType := Real" } GE_Contact(in1 := #tempReal, in2 := "DrillTorqSetMax")
      Coil( "DrillTorqLimited" )
   END_RUNG
   RUNG wire#powerrail
      Mul(in1 := "MUTorqSetFtLbs", in2 := "Settings".TorqSetFactor, out => #tempReal)
      Div(in1 := #tempReal, in2 := "Settings".TorqOutLSHT, out => "MUTorqSetPSI")
      Add(in1 := "MUTorqSetPSI", in2 := "Settings".TorqOutExtraPSI, out => "MUTorqSetPSI")
      { S7_Templates := "value_type := Real" } Limit(mn := "Settings".TorqOutMinPSI, in := "MUTorqSetPSI", mx := "Settings".TorqOutMaxPSI, out => "MUTorqSetPSI")
   END_RUNG
   RUNG wire#powerrail
      I_Contact( "HSLT_Sol" )
      Mul(in1 := "DrillTorqSetFtLbs", in2 := "Settings".TorqSetFactor, out => #tempReal)
      Div(in1 := #tempReal, in2 := "Settings".TorqOutLSHT, out => "DrillTorqSetPSI")
      Add(in1 := "DrillTorqSetPSI", in2 := "Settings".TorqOutExtraPSI, out => "DrillTorqSetPSI")
      { S7_Templates := "value_type := Real" } Limit(mn := "Settings".TorqOutMinPSI, in := "DrillTorqSetPSI", mx := "Settings".TorqOutMaxPSI, out => "DrillTorqSetPSI")
   END_RUNG
   RUNG wire#powerrail
      Contact( "HSLT_Sol" )
      Mul(in1 := "DrillTorqSetFtLbs", in2 := "Settings".TorqSetFactor, out => #tempReal)
      Div(in1 := #tempReal, in2 := "Settings".TorqOutHSLT, out => "DrillTorqSetPSI")
      Add(in1 := "DrillTorqSetPSI", in2 := "Settings".TorqOutExtraPSI, out => "DrillTorqSetPSI")
      { S7_Templates := "value_type := Real" } Limit(mn := "Settings".TorqOutMinPSI, in := "DrillTorqSetPSI", mx := "Settings".TorqOutMaxPSI, out => "DrillTorqSetPSI")
   END_RUNG
   RUNG wire#powerrail
      Div(in1 := "Settings".MUDoneTHper, in2 := 100.0, out => #tempReal)
      Mul(in1 := "MUTorqSetFtLbs", in2 := #tempReal, out => "MUDoneSetFtLbs")
   END_RUNG
   // the same network as SCL:
   #tempReal := "MUTorqPotPerFilt" / 100.0;
   "MUTorqSetFtLbs" := #tempReal * "Settings".TorqPotMaxFtLbs;
   "DrillTorqSetMax" := "MUTorqSetFtLbs" * 0.95;
   "MUTorqSetKFtLbs" := "MUTorqSetFtLbs" / 1000.0;
   #tempReal := "DrillTorqPotPerFilt" / 100.0;
   #tempReal := #tempReal * "Settings".TorqPotMaxFtLbs;
   "DrillTorqSetFtLbs" := LIMIT(MN := 0.0, IN := #tempReal, MX := "DrillTorqSetMax");
   "DrillTorqSetKFtLbs" := "DrillTorqSetFtLbs" / 1000.0;
   "DrillTorqLimited" := #tempReal >= "DrillTorqSetMax";
   #tempReal := "MUTorqSetFtLbs" * "Settings".TorqSetFactor;
   "MUTorqSetPSI" := #tempReal / "Settings".TorqOutLSHT;
   "MUTorqSetPSI" := "MUTorqSetPSI" + "Settings".TorqOutExtraPSI;
   "MUTorqSetPSI" := LIMIT(MN := "Settings".TorqOutMinPSI, IN := "MUTorqSetPSI", MX := "Settings".TorqOutMaxPSI);
   IF NOT "HSLT_Sol" THEN
       #tempReal := "DrillTorqSetFtLbs" * "Settings".TorqSetFactor;
       "DrillTorqSetPSI" := #tempReal / "Settings".TorqOutLSHT;
       "DrillTorqSetPSI" := "DrillTorqSetPSI" + "Settings".TorqOutExtraPSI;
       "DrillTorqSetPSI" := LIMIT(MN := "Settings".TorqOutMinPSI, IN := "DrillTorqSetPSI", MX := "Settings".TorqOutMaxPSI);
   END_IF;
   IF "HSLT_Sol" THEN
       #tempReal := "DrillTorqSetFtLbs" * "Settings".TorqSetFactor;
       "DrillTorqSetPSI" := #tempReal / "Settings".TorqOutHSLT;
       "DrillTorqSetPSI" := "DrillTorqSetPSI" + "Settings".TorqOutExtraPSI;
       "DrillTorqSetPSI" := LIMIT(MN := "Settings".TorqOutMinPSI, IN := "DrillTorqSetPSI", MX := "Settings".TorqOutMaxPSI);
   END_IF;
   #tempReal := "Settings".MUDoneTHper / 100.0;
   "MUDoneSetFtLbs" := "MUTorqSetFtLbs" * #tempReal;
END_REGION

REGION Network 8: Auto Makeup Torq Setpoints
   // These setpoints are based on a percent of the user input
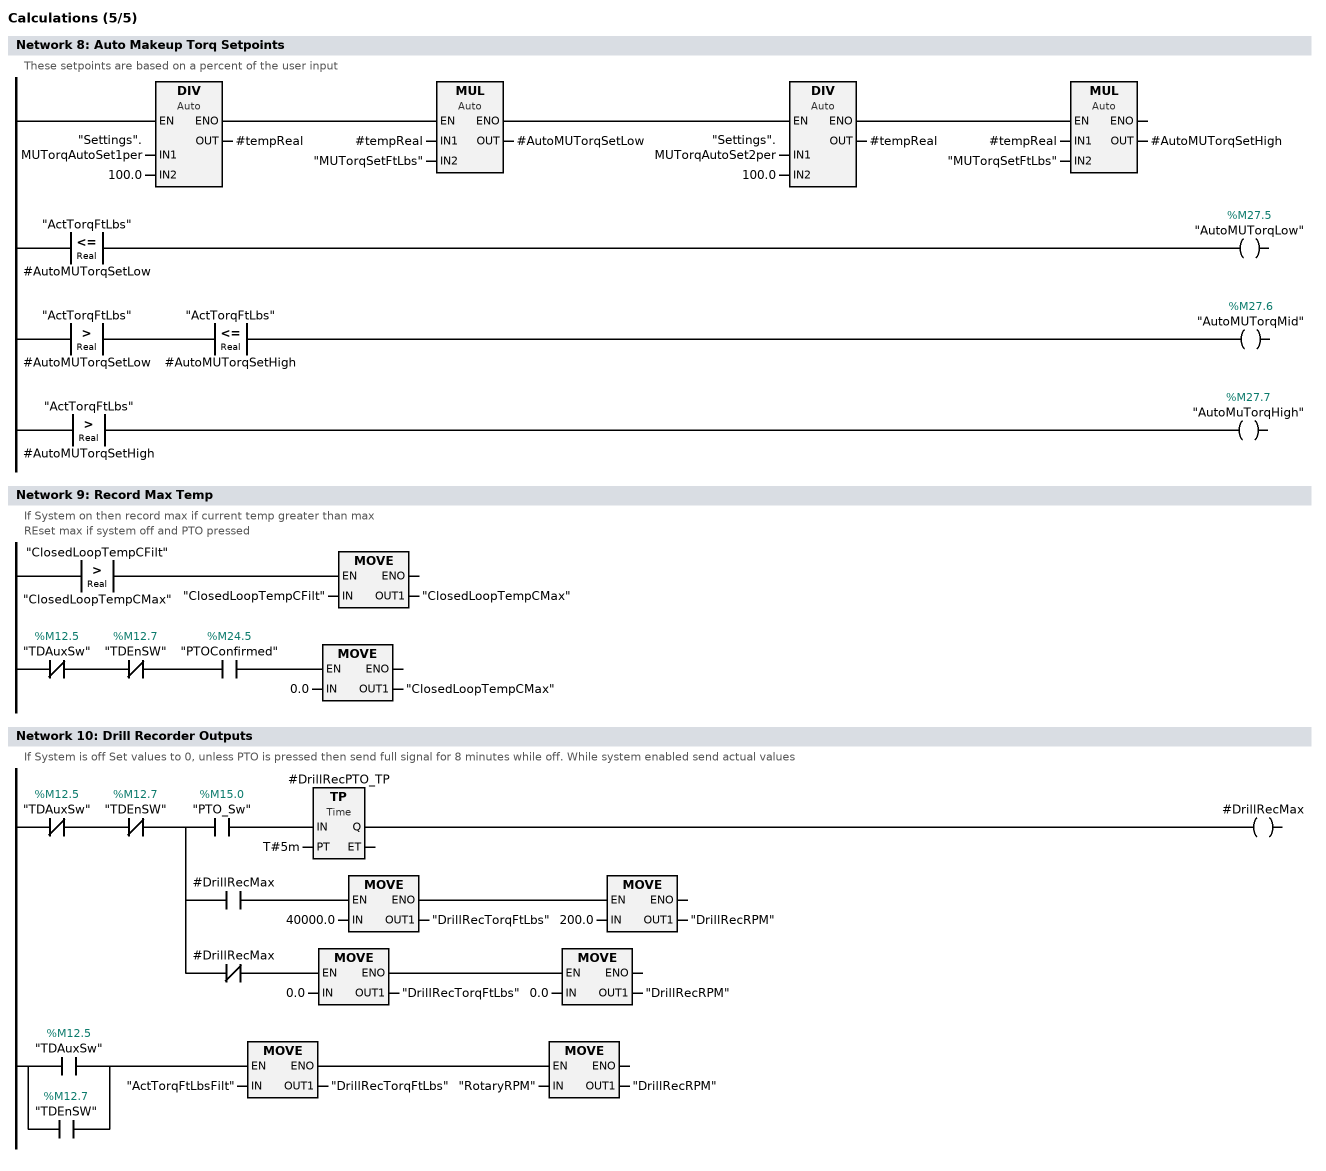
   RUNG wire#powerrail
      Div(in1 := "Settings".MUTorqAutoSet1per, in2 := 100.0, out => #tempReal)
      Mul(in1 := #tempReal, in2 := "MUTorqSetFtLbs", out => #AutoMUTorqSetLow)
      Div(in1 := "Settings".MUTorqAutoSet2per, in2 := 100.0, out => #tempReal)
      Mul(in1 := #tempReal, in2 := "MUTorqSetFtLbs", out => #AutoMUTorqSetHigh)
   END_RUNG
   RUNG wire#powerrail
      { S7_Templates := "SrcType := Real" } LE_Contact(in1 := "ActTorqFtLbs", in2 := #AutoMUTorqSetLow)
      Coil( "AutoMUTorqLow" )
   END_RUNG
   RUNG wire#powerrail
      { S7_Templates := "SrcType := Real" } GT_Contact(in1 := "ActTorqFtLbs", in2 := #AutoMUTorqSetLow)
      { S7_Templates := "SrcType := Real" } LE_Contact(in1 := "ActTorqFtLbs", in2 := #AutoMUTorqSetHigh)
      Coil( "AutoMUTorqMid" )
   END_RUNG
   RUNG wire#powerrail
      { S7_Templates := "SrcType := Real" } GT_Contact(in1 := "ActTorqFtLbs", in2 := #AutoMUTorqSetHigh)
      Coil( "AutoMuTorqHigh" )
   END_RUNG
   // the same network as SCL:
   #tempReal := "Settings".MUTorqAutoSet1per / 100.0;
   #AutoMUTorqSetLow := #tempReal * "MUTorqSetFtLbs";
   #tempReal := "Settings".MUTorqAutoSet2per / 100.0;
   #AutoMUTorqSetHigh := #tempReal * "MUTorqSetFtLbs";
   "AutoMUTorqLow" := "ActTorqFtLbs" <= #AutoMUTorqSetLow;
   "AutoMUTorqMid" := ("ActTorqFtLbs" > #AutoMUTorqSetLow) AND ("ActTorqFtLbs" <= #AutoMUTorqSetHigh);
   "AutoMuTorqHigh" := "ActTorqFtLbs" > #AutoMUTorqSetHigh;
END_REGION

REGION Network 9: Record Max Temp
   // If System on then record max if current temp greater than max
   // REset max if system off and PTO pressed
   RUNG wire#powerrail
      { S7_Templates := "SrcType := Real" } GT_Contact(in1 := "ClosedLoopTempCFilt", in2 := "ClosedLoopTempCMax")
      Move(in := "ClosedLoopTempCFilt", out1 => "ClosedLoopTempCMax")
   END_RUNG
   RUNG wire#powerrail
      I_Contact( "TDAuxSw" )
      I_Contact( "TDEnSW" )
      Contact( "PTOConfirmed" )
      Move(in := 0.0, out1 => "ClosedLoopTempCMax")
   END_RUNG
   // the same network as SCL:
   IF "ClosedLoopTempCFilt" > "ClosedLoopTempCMax" THEN
       "ClosedLoopTempCMax" := "ClosedLoopTempCFilt";
   END_IF;
   IF NOT "TDAuxSw" AND NOT "TDEnSW" AND "PTOConfirmed" THEN "ClosedLoopTempCMax" := 0.0; END_IF;
END_REGION

REGION Network 10: Drill Recorder Outputs
   // If System is off Set values to 0, unless PTO is pressed then send full signal for 8 minutes while off. While system enabled send actual values
   RUNG wire#powerrail
      I_Contact( "TDAuxSw" )
      I_Contact( "TDEnSW" )
      wire#w1
      Contact( "PTO_Sw" )
      { S7_Templates := "time_type := Time" } #DrillRecPTO_TP.TP(pt := T#5m, et =>)
      Coil( #DrillRecMax )
   END_RUNG
   RUNG wire#w1
      Contact( #DrillRecMax )
      Move(in := 40000.0, out1 => "DrillRecTorqFtLbs")
      Move(in := 200.0, out1 => "DrillRecRPM")
   END_RUNG
   RUNG wire#w1
      I_Contact( #DrillRecMax )
      Move(in := 0.0, out1 => "DrillRecTorqFtLbs")
      Move(in := 0.0, out1 => "DrillRecRPM")
   END_RUNG
   RUNG wire#powerrail
      Contact( "TDAuxSw" )
      wire#w2
      Move(in := "ActTorqFtLbsFilt", out1 => "DrillRecTorqFtLbs")
      Move(in := "RotaryRPM", out1 => "DrillRecRPM")
   END_RUNG
   RUNG wire#powerrail
      Contact( "TDEnSW" )
   END_RUNG wire#w2
   // the same network as SCL:
   #_w1 := NOT "TDAuxSw" AND NOT "TDEnSW";
   #DrillRecPTO_TP(IN := #_w1 AND "PTO_Sw", PT := T#5m);   // TP
   #DrillRecMax := #DrillRecPTO_TP.Q;
   IF #_w1 AND #DrillRecMax THEN
       "DrillRecTorqFtLbs" := 40000.0;
       "DrillRecRPM" := 200.0;
   END_IF;
   IF #_w1 AND NOT #DrillRecMax THEN
       "DrillRecTorqFtLbs" := 0.0;
       "DrillRecRPM" := 0.0;
   END_IF;
   IF "TDAuxSw" OR "TDEnSW" THEN
       "DrillRecTorqFtLbs" := "ActTorqFtLbsFilt";
       "DrillRecRPM" := "RotaryRPM";
   END_IF;
END_REGION
END_FUNCTION_BLOCK

FUNCTION_BLOCK "Rot_Pos_Calc"
{ S7_Optimized_Access := 'TRUE' }
VERSION : 0.1
   VAR_INPUT 
      PulsesPerRev : Int;   // Encoder pulses per revolutions. 
      Counts : DInt;   // Encoder counts
      UL_OF : Bool;   // Counter Upper Limit Overflow
      LL_OF : Bool;   // Counter Lower Limit Over Flow
      StoppedTime : Time := T#2s;   // Time without a encoder feedback to says system is stopped/not moving
      RolloverValue : LReal;
   END_VAR

   VAR_OUTPUT 
      RotPosAbsDeg : Real;
      RotPosRelDeg : Real := 0.0;
      RotTurns : Real;
      Stopped : Bool;
      DirFwd : Bool;
      DirRev : Bool;
      DegPerCount : Real;
   END_VAR

   VAR_IN_OUT 
      ZeroPos : Bool;   // Used to Reset Position to zero. Flag will reset to zero once position is zero
      LDSlot0_1 : Byte;   // Upper 4 Bits LD SLot 1 and lower 4 BITS to load Slot0 
      Slot0 : Real;
      Slot1 : Real;
   END_VAR

   VAR 
      PosAbsDegLReal : LReal := 0.0;
      Static_1 : Real;
      LastEncCount : DInt;
      Stopped_TON {InstructionName := 'TON_TIME'; LibVersion := '1.0'} : TON_TIME;
   END_VAR

   VAR_TEMP 
      PulsesPerRevAdj : Int;
   END_VAR


BEGIN
	(* #RotPosCalc Written BY Kristopher Gimenez January 23,2023
	This block is used to to calculate actual rotary position, stopped status and direction of the rotary position.
	Note that position is always counted from 0 as counter is reset when zero position selected.
	*)
	
	
	//Encoder rotary position
	// 2*PPR = counts per Rev = 360. Counter rollover at 2147483647 to - 2147483647
	IF "HMI_DB".OscTurnFwd <= 1 OR "HMI_DB".OscTurnRev <= 1 THEN
	    #PulsesPerRevAdj := 22;
	ELSIF "HMI_DB".OscTurnFwd <= 2 OR "HMI_DB".OscTurnRev <= 2 THEN
	    #PulsesPerRevAdj := 22;
	ELSIF "HMI_DB".OscTurnFwd <= 3 OR "HMI_DB".OscTurnRev <= 3 THEN
	    #PulsesPerRevAdj := 22;
	ELSIF "HMI_DB".OscTurnFwd <= 4 OR "HMI_DB".OscTurnRev <= 4 THEN
	    #PulsesPerRevAdj := 22;
	ELSE
	    #PulsesPerRevAdj := 22;
	END_IF;
	
	#Static_1 := 360.0/INT_TO_REAL(#PulsesPerRevAdj) ;
	#DegPerCount := #Static_1;
	
	IF #UL_OF THEN //if overflow over the top limit, count from neg limit and add upper range
	    #PosAbsDegLReal := DINT_TO_LREAL(LREAL_TO_DINT(-#RolloverValue) - #Counts)*#Static_1 + LREAL_TO_DINT(#RolloverValue * #Static_1);
	ELSIF #LL_OF THEN //if overflow over the bottom limit, count from pos limit and add lower range
	    #PosAbsDegLReal := DINT_TO_LREAL(LREAL_TO_DINT(#RolloverValue) - #Counts)*#Static_1  + LREAL_TO_DINT(#RolloverValue* #Static_1);
	ELSE //no overflow 15deg/count
	    #PosAbsDegLReal := DINT_TO_LREAL(#Counts) * #Static_1;
	END_IF;
	
	#RotPosAbsDeg := LREAL_TO_REAL(#PosAbsDegLReal);
	#RotPosRelDeg := DINT_TO_REAL(LREAL_TO_DINT(#PosAbsDegLReal) MOD 360);
	#RotTurns := LREAL_TO_REAL(#PosAbsDegLReal/360.0);
	
	
	//Use this load request to specify the meaning of the value in SLOT_m:
	(*
	• 0000B means: No action, idle
	• 0001B means: Load counter value
	• 0010B not permitted
	• 0011B means: Load start value
	• 0100B means: Load comparison value 0
	• 0101B means: Load comparison value 1
	• 0110B means: Load counting low limit
	• 0111B means: Load counting high limit*)
	
	IF #ZeroPos AND (#Counts <> 0) THEN //if zero request received and position is not zero.
	    #Slot0 := 0; // set value to load to zero
	    #LDSlot0_1 := 1; //load slot 0.
	    "SwitchSWGATE" := 0;
	ELSIF #ZeroPos AND (#Counts = 0) THEN //position has been reset. Reset load variable and position reset
	    #LDSlot0_1 := 0;//don't load anything
	    #ZeroPos := 0;
	    "SwitchSWGATE" := 1;
	ELSE //reset slot load
	    #LDSlot0_1 := 0;//don't load anything
	    "SwitchSWGATE" := 1;
	END_IF;
	
	//IF counts = last counts for set time. Movement stopped. 
	
	#Stopped_TON(IN:=(#Counts=#LastEncCount),
	             PT:=#StoppedTime,
	             Q => #Stopped);
	
	IF #Stopped THEN
	    #DirFwd := 0;
	    #DirRev := 0;
	    "RotaryStopped" := 1;
	ELSIF #Counts < #LastEncCount THEN
	    #DirFwd := 0;
	    #DirRev := 1;
	    "RotaryStopped" := 0;
	ELSIF #Counts > #LastEncCount THEN
	    #DirFwd := 1;
	    #DirRev := 0;
	    "RotaryStopped" := 0;
	END_IF;
	
	IF #RotPosRelDeg >= 0 THEN
	    "RotRelPosDegHMIPos" := #RotPosRelDeg;
	ELSE
	    "RotRelPosDegHMIPos" := 360.0 + #RotPosRelDeg;
	END_IF;
	
	IF "HMI_DB".OscHomeRelDeg >= 0 THEN
	    "OscHomeRelDegHMIPos" := "HMI_DB".OscHomeRelDeg;
	ELSE
	    "OscHomeRelDegHMIPos" := 360.0 + "HMI_DB".OscHomeRelDeg;
	END_IF;
	
	
	    "RotaryRPMHMI" := ABS ("RotaryRPM");
	    #LastEncCount := #Counts;
	
	
	
	
END_FUNCTION_BLOCK

FUNCTION "Ai_Scale0_10V" : Void
{ S7_Optimized_Access := 'TRUE' }
VERSION : 0.1
   VAR_INPUT 
      VoltInput : Real;   // 0-10 Volt Input
      OutMin : Real;
      OutMax : Real;
   END_VAR

   VAR_OUTPUT 
      OutScaledReal : Real;
   END_VAR


BEGIN
	(* Ai_Scale0_10V Written BY Kristopher Gimenez January 24,2023
	This block is used to convert a 0-10mA input to a scaled output based on input Min and Max
	*)
	
	
	#OutScaledReal := (#"VoltInput"/ 10 * (#OutMax - #OutMin)) + #OutMin;
	
	
	
	
END_FUNCTION

FUNCTION "Ai_Scale420mA" : Void
{ S7_Optimized_Access := 'TRUE' }
VERSION : 0.1
   VAR_INPUT 
      "420mAInput" : Real;
      OutMin : Real;
      OutMax : Real;
   END_VAR

   VAR_OUTPUT 
      OutScaledReal : Real;
   END_VAR


BEGIN
	(* Ai_Scale420mA Written BY Kristopher Gimenez January 24,2023
	This block is used to convert a 4-20mA input to a scaled output based on input Min and Max
	*)
	
	
	#OutScaledReal := ((#"420mAInput" - 4) / 16 * (#OutMax - #OutMin)) + #OutMin;
	
	
	
	
END_FUNCTION

FUNCTION "F_To_C_Convert" : Void
{ S7_Optimized_Access := 'TRUE' }
VERSION : 0.1
   VAR_INPUT 
      Fdegree : Real;
   END_VAR

   VAR_OUTPUT 
      Cdegree : Real;
   END_VAR


BEGIN
	#Cdegree := (#Fdegree - 32.0) * 5 / 9.0;
END_FUNCTION

FUNCTION_BLOCK "LowPassFilter"
{ S7_Optimized_Access := 'TRUE' }
VERSION : 0.1
   VAR_INPUT 
      InputSignal : Real;
      Alpha : Real;
   END_VAR

   VAR_OUTPUT 
      FilteredSignal : Real;
   END_VAR

   VAR 
      LastValue : Real;
      AlphaInt : Real;   // Internal Alpha within scaling range
   END_VAR


BEGIN
	(* #LowPassFilter Written BY Kristopher Gimenez January 23,2023
	This block is used to as a First Order Low Pass Filter  (same as Exponentially Weighted Moving Average Filter)
	
	Alpha  must be >= 0 and < 1
	
	set Alpha to 0.0 for no filtering
	
	FilteredSignal = alpha*lastFiltered +(1-Alpha) * Signal
	*)
	
	IF #Alpha < 0.0 THEN
	    #AlphaInt := 0;
	ELSIF #Alpha > 1.0 THEN
	    #AlphaInt := 1.0;
	ELSE
	    #AlphaInt := #Alpha;
	END_IF;
	
	#FilteredSignal := #AlphaInt * #LastValue +(1-#AlphaInt) * #InputSignal;
	#LastValue := #FilteredSignal;
	
	
END_FUNCTION_BLOCK

FUNCTION "Pump_Output" : Void
{ S7_Optimized_Access := 'TRUE' }
VERSION : 0.1
   VAR_INPUT 
      Disable : Bool;   // Enable the Block to convert. Otherwise output set to min
      InputValue : Real;
      InMin : Real;
      InMax : Real;
      OutMin_mA : Real;
      OutMax_mA : Real;
   END_VAR

   VAR_OUTPUT 
      mAOut : Real;
   END_VAR


BEGIN
	(* Pump_Output Written BY Kristopher Gimenez January 19,2023
	This block will will convert and scale an input to output for the pump control
	*)
	
	
	
	IF #InputValue <= #InMin OR #Disable THEN //if input less than min or not enabled set output to min
	    #mAOut := #OutMin_mA;
	ELSIF #InputValue >= #InMax THEN//if input greater than amx set output to max
	    #mAOut := #OutMax_mA;
	ELSE//else input in range so scale.
	    #mAOut := ((#InputValue - #InMin) / (#InMax - #InMin) * (#OutMax_mA - #OutMin_mA)) + #OutMin_mA;
	END_IF;
	
	
END_FUNCTION

FUNCTION_BLOCK "Aux_Motor_Control"   // FB12, LAD
{ S7_Optimized_Access := 'TRUE' }
// Written BY Kristopher Gimenez January 25,2023
// This block is used to control the Aux, and Cooler fan motors.
// stored: AutoNumber false, MemoryReserve 100, SetENOAutomatically false
   VAR
      AuxPumpStartTOF { S7_SetPoint := 'True'} : TOF_TIME;
      AuxPumpFailTON { S7_SetPoint := 'True'} : TON_TIME;
      CoolingFanFailTON { S7_SetPoint := 'True'} : TON_TIME;
      CoolingFanStartTON { S7_SetPoint := 'True'} : TOF_TIME;
   END_VAR
BEGIN

REGION Network 1: Aux Pump Start
   // TOFF used on Aux pump allows 2 seconds for functions to stop when system is disabled before pump is shutdown and to maintain while switching between Aux and TD Enabled
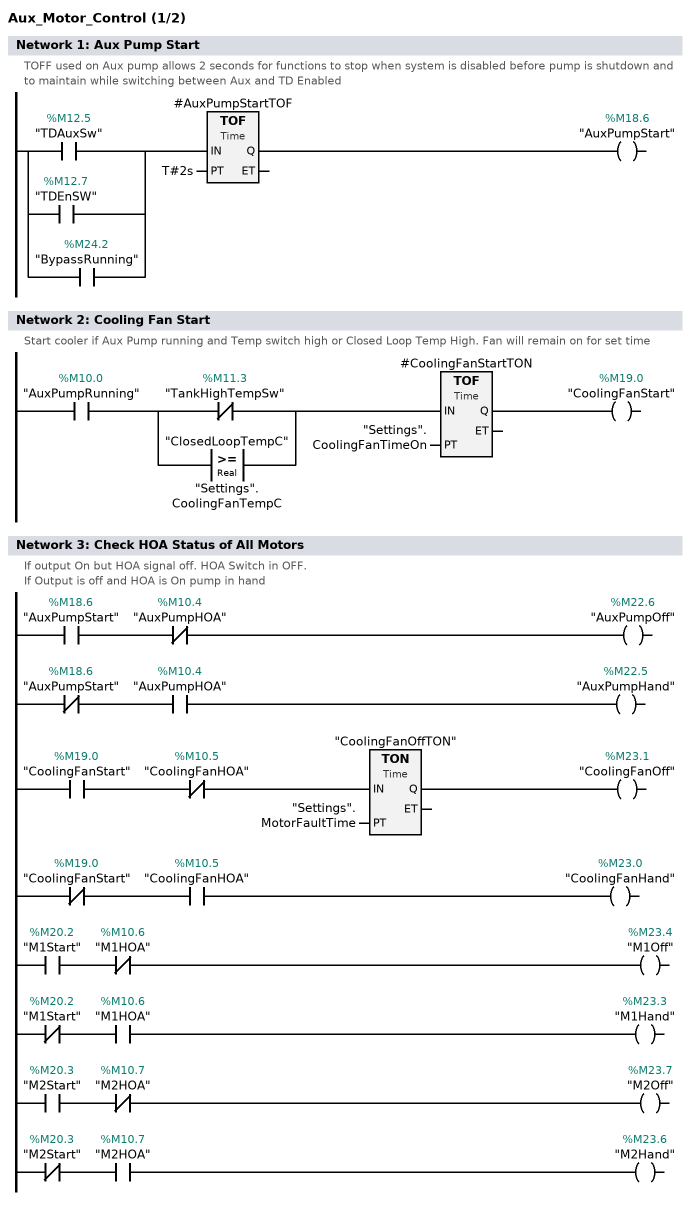
   RUNG wire#powerrail
      Contact( "TDAuxSw" )
      wire#w1
      { S7_Templates := "time_type := Time" } #AuxPumpStartTOF.TOF(pt := T#2s, et =>)
      Coil( "AuxPumpStart" )
   END_RUNG
   RUNG wire#powerrail
      Contact( "TDEnSW" )
   END_RUNG wire#w1
   RUNG wire#powerrail
      Contact( "BypassRunning" )
   END_RUNG wire#w1
   // the same network as SCL:
   #AuxPumpStartTOF(IN := "TDAuxSw" OR "TDEnSW" OR "BypassRunning", PT := T#2s);   // TOF
   "AuxPumpStart" := #AuxPumpStartTOF.Q;
END_REGION

REGION Network 2: Cooling Fan Start
   // Start cooler if Aux Pump running and Temp switch high or Closed Loop Temp High. Fan will remain on for set time
   RUNG wire#powerrail
      Contact( "AuxPumpRunning" )
      wire#w1
      I_Contact( "TankHighTempSw" )
      wire#w2
      { S7_Templates := "time_type := Time" } #CoolingFanStartTON.TOF(pt := "Settings".CoolingFanTimeOn, et =>)
      Coil( "CoolingFanStart" )
   END_RUNG
   RUNG wire#w1
      { S7_Templates := "SrcType := Real" } GE_Contact(in1 := "ClosedLoopTempC", in2 := "Settings".CoolingFanTempC)
   END_RUNG wire#w2
   // the same network as SCL:
   #CoolingFanStartTON(IN := "AuxPumpRunning" AND (NOT "TankHighTempSw" OR ("ClosedLoopTempC" >= "Settings".CoolingFanTempC)),   // TOF
                       PT := "Settings".CoolingFanTimeOn);
   "CoolingFanStart" := #CoolingFanStartTON.Q;
END_REGION

REGION Network 3: Check HOA Status of All Motors
   // If output On but HOA signal off. HOA Switch in OFF. 
   // If Output is off and HOA is On pump in hand
   RUNG wire#powerrail
      Contact( "AuxPumpStart" )
      I_Contact( "AuxPumpHOA" )
      Coil( "AuxPumpOff" )
   END_RUNG
   RUNG wire#powerrail
      I_Contact( "AuxPumpStart" )
      Contact( "AuxPumpHOA" )
      Coil( "AuxPumpHand" )
   END_RUNG
   RUNG wire#powerrail
      Contact( "CoolingFanStart" )
      I_Contact( "CoolingFanHOA" )
      { S7_Templates := "time_type := Time" } "CoolingFanOffTON".TON(pt := "Settings".MotorFaultTime, et =>)
      Coil( "CoolingFanOff" )
   END_RUNG
   RUNG wire#powerrail
      I_Contact( "CoolingFanStart" )
      Contact( "CoolingFanHOA" )
      Coil( "CoolingFanHand" )
   END_RUNG
   RUNG wire#powerrail
      Contact( "M1Start" )
      I_Contact( "M1HOA" )
      Coil( "M1Off" )
   END_RUNG
   RUNG wire#powerrail
      I_Contact( "M1Start" )
      Contact( "M1HOA" )
      Coil( "M1Hand" )
   END_RUNG
   RUNG wire#powerrail
      Contact( "M2Start" )
      I_Contact( "M2HOA" )
      Coil( "M2Off" )
   END_RUNG
   RUNG wire#powerrail
      I_Contact( "M2Start" )
      Contact( "M2HOA" )
      Coil( "M2Hand" )
   END_RUNG
   // the same network as SCL:
   "AuxPumpOff" := "AuxPumpStart" AND NOT "AuxPumpHOA";
   "AuxPumpHand" := NOT "AuxPumpStart" AND "AuxPumpHOA";
   "CoolingFanOffTON".TON(IN := "CoolingFanStart" AND NOT "CoolingFanHOA", PT := "Settings".MotorFaultTime);
   "CoolingFanOff" := "CoolingFanOffTON".Q;
   "CoolingFanHand" := NOT "CoolingFanStart" AND "CoolingFanHOA";
   "M1Off" := "M1Start" AND NOT "M1HOA";
   "M1Hand" := NOT "M1Start" AND "M1HOA";
   "M2Off" := "M2Start" AND NOT "M2HOA";
   "M2Hand" := NOT "M2Start" AND "M2HOA";
END_REGION

REGION Network 4: Motor Starter Fault Status
   // If pump start signal seen on HOA input but it has not started by fault time. Set motor fault
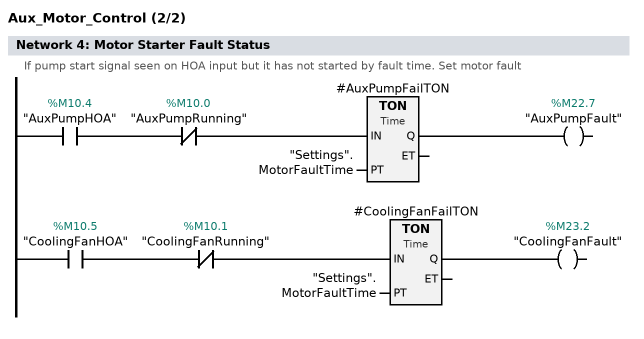
   RUNG wire#powerrail
      Contact( "AuxPumpHOA" )
      I_Contact( "AuxPumpRunning" )
      { S7_Templates := "time_type := Time" } #AuxPumpFailTON.TON(pt := "Settings".MotorFaultTime, et =>)
      Coil( "AuxPumpFault" )
   END_RUNG
   RUNG wire#powerrail
      Contact( "CoolingFanHOA" )
      I_Contact( "CoolingFanRunning" )
      { S7_Templates := "time_type := Time" } #CoolingFanFailTON.TON(pt := "Settings".MotorFaultTime, et =>)
      Coil( "CoolingFanFault" )
   END_RUNG
   // the same network as SCL:
   #AuxPumpFailTON(IN := "AuxPumpHOA" AND NOT "AuxPumpRunning", PT := "Settings".MotorFaultTime);   // TON
   "AuxPumpFault" := #AuxPumpFailTON.Q;
   #CoolingFanFailTON(IN := "CoolingFanHOA" AND NOT "CoolingFanRunning", PT := "Settings".MotorFaultTime);   // TON
   "CoolingFanFault" := #CoolingFanFailTON.Q;
END_REGION
END_FUNCTION_BLOCK

FUNCTION_BLOCK "TD_Motor_Start_Elec"   // FB13, LAD
{ S7_Optimized_Access := 'TRUE' }
// Written BY Kristopher Gimenez January 25,2023
// This block is used to control the TD motors on an Elec HPUs
// stored: AutoNumber false, MemoryReserve 100, SetENOAutomatically false
   VAR
      TDP1FailTON { S7_SetPoint := 'True'} : TON_TIME;
      TDP2FailTON { S7_SetPoint := 'True'} : TON_TIME;
   END_VAR
BEGIN

REGION Network 1: Enable Top Drive
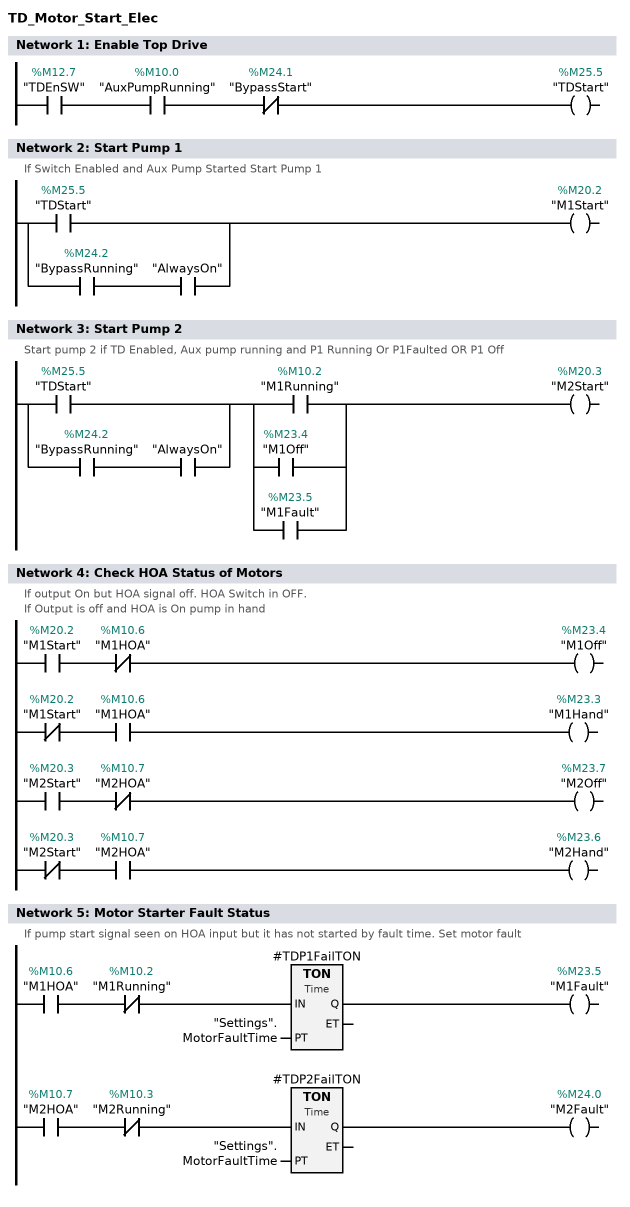
   RUNG wire#powerrail
      Contact( "TDEnSW" )
      Contact( "AuxPumpRunning" )
      I_Contact( "BypassStart" )
      Coil( "TDStart" )
   END_RUNG
   // the same network as SCL:
   "TDStart" := "TDEnSW" AND "AuxPumpRunning" AND NOT "BypassStart";
END_REGION

REGION Network 2: Start Pump 1
   // If Switch Enabled and Aux Pump Started Start Pump 1
   RUNG wire#powerrail
      Contact( "TDStart" )
      wire#w1
      Coil( "M1Start" )
   END_RUNG
   RUNG wire#powerrail
      Contact( "BypassRunning" )
      Contact( "AlwaysOn" )
   END_RUNG wire#w1
   // the same network as SCL:
   "M1Start" := "TDStart" OR ("BypassRunning" AND "AlwaysOn");
END_REGION

REGION Network 3: Start Pump 2
   // Start pump 2 if TD Enabled, Aux pump running and P1 Running Or P1Faulted OR P1 Off
   RUNG wire#powerrail
      Contact( "TDStart" )
      wire#w1
      Contact( "M1Running" )
      wire#w2
      Coil( "M2Start" )
   END_RUNG
   RUNG wire#powerrail
      Contact( "BypassRunning" )
      Contact( "AlwaysOn" )
   END_RUNG wire#w1
   RUNG wire#w1
      Contact( "M1Off" )
   END_RUNG wire#w2
   RUNG wire#w1
      Contact( "M1Fault" )
   END_RUNG wire#w2
   // the same network as SCL:
   "M2Start" := ("TDStart" OR ("BypassRunning" AND "AlwaysOn")) AND ("M1Running" OR "M1Off" OR "M1Fault");
END_REGION

REGION Network 4: Check HOA Status of Motors
   // If output On but HOA signal off. HOA Switch in OFF. 
   // If Output is off and HOA is On pump in hand
   RUNG wire#powerrail
      Contact( "M1Start" )
      I_Contact( "M1HOA" )
      Coil( "M1Off" )
   END_RUNG
   RUNG wire#powerrail
      I_Contact( "M1Start" )
      Contact( "M1HOA" )
      Coil( "M1Hand" )
   END_RUNG
   RUNG wire#powerrail
      Contact( "M2Start" )
      I_Contact( "M2HOA" )
      Coil( "M2Off" )
   END_RUNG
   RUNG wire#powerrail
      I_Contact( "M2Start" )
      Contact( "M2HOA" )
      Coil( "M2Hand" )
   END_RUNG
   // the same network as SCL:
   "M1Off" := "M1Start" AND NOT "M1HOA";
   "M1Hand" := NOT "M1Start" AND "M1HOA";
   "M2Off" := "M2Start" AND NOT "M2HOA";
   "M2Hand" := NOT "M2Start" AND "M2HOA";
END_REGION

REGION Network 5: Motor Starter Fault Status
   // If pump start signal seen on HOA input but it has not started by fault time. Set motor fault
   RUNG wire#powerrail
      Contact( "M1HOA" )
      I_Contact( "M1Running" )
      { S7_Templates := "time_type := Time" } #TDP1FailTON.TON(pt := "Settings".MotorFaultTime, et =>)
      Coil( "M1Fault" )
   END_RUNG
   RUNG wire#powerrail
      Contact( "M2HOA" )
      I_Contact( "M2Running" )
      { S7_Templates := "time_type := Time" } #TDP2FailTON.TON(pt := "Settings".MotorFaultTime, et =>)
      Coil( "M2Fault" )
   END_RUNG
   // the same network as SCL:
   #TDP1FailTON(IN := "M1HOA" AND NOT "M1Running", PT := "Settings".MotorFaultTime);   // TON
   "M1Fault" := #TDP1FailTON.Q;
   #TDP2FailTON(IN := "M2HOA" AND NOT "M2Running", PT := "Settings".MotorFaultTime);   // TON
   "M2Fault" := #TDP2FailTON.Q;
END_REGION
END_FUNCTION_BLOCK

FUNCTION_BLOCK "TD_Motor_Start_CAT"   // FB14, LAD
{ S7_Optimized_Access := 'TRUE' }
// Written BY Kristopher Gimenez January 25,2023
// This block is used to control the Aux, and Cooler fan motors.
// stored: AutoNumber false, MemoryReserve 100, SetENOAutomatically false
   VAR
      EngineFault_TON { S7_SetPoint := 'True'} : TON_TIME;
   END_VAR
   VAR_TEMP
      tempReal : Real;
   END_VAR
BEGIN

REGION Network 1: Engine Speed
   // Pulse Per Second X 60sc/m /PPR
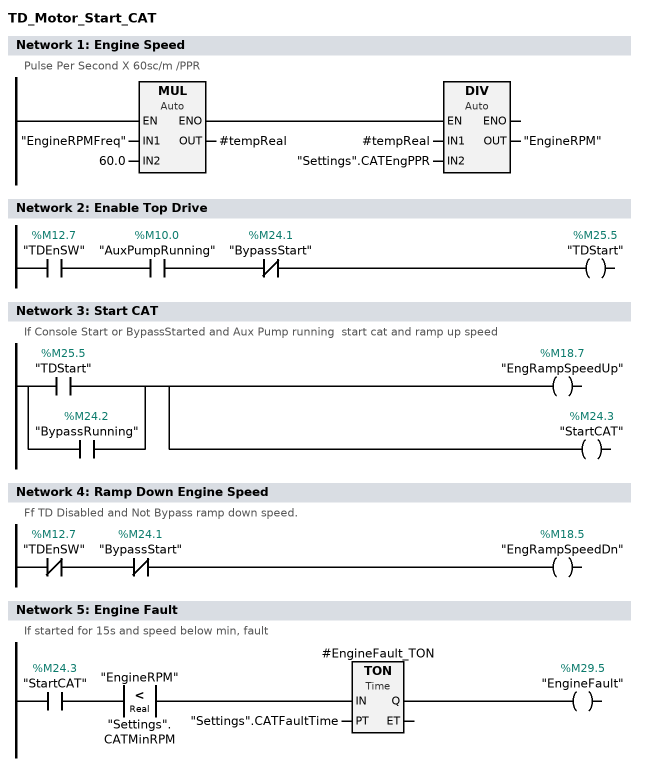
   RUNG wire#powerrail
      Mul(in1 := "EngineRPMFreq", in2 := 60.0, out => #tempReal)
      Div(in1 := #tempReal, in2 := "Settings".CATEngPPR, out => "EngineRPM")
   END_RUNG
   // the same network as SCL:
   #tempReal := "EngineRPMFreq" * 60.0;
   "EngineRPM" := #tempReal / "Settings".CATEngPPR;
END_REGION

REGION Network 2: Enable Top Drive
   RUNG wire#powerrail
      Contact( "TDEnSW" )
      Contact( "AuxPumpRunning" )
      I_Contact( "BypassStart" )
      Coil( "TDStart" )
   END_RUNG
   // the same network as SCL:
   "TDStart" := "TDEnSW" AND "AuxPumpRunning" AND NOT "BypassStart";
END_REGION

REGION Network 3: Start CAT
   // If Console Start or BypassStarted and Aux Pump running  start cat and ramp up speed
   RUNG wire#powerrail
      Contact( "TDStart" )
      wire#w1
      Coil( "EngRampSpeedUp" )
   END_RUNG
   RUNG wire#powerrail
      Contact( "BypassRunning" )
   END_RUNG wire#w1
   RUNG wire#w1
      Coil( "StartCAT" )
   END_RUNG
   // the same network as SCL:
   "EngRampSpeedUp" := "TDStart" OR "BypassRunning";
   "StartCAT" := "EngRampSpeedUp";
END_REGION

REGION Network 4: Ramp Down Engine Speed
   // Ff TD Disabled and Not Bypass ramp down speed.
   RUNG wire#powerrail
      I_Contact( "TDEnSW" )
      I_Contact( "BypassStart" )
      Coil( "EngRampSpeedDn" )
   END_RUNG
   // the same network as SCL:
   "EngRampSpeedDn" := NOT "TDEnSW" AND NOT "BypassStart";
END_REGION

REGION Network 5: Engine Fault
   // If started for 15s and speed below min, fault
   RUNG wire#powerrail
      Contact( "StartCAT" )
      { S7_Templates := "SrcType := Real" } LT_Contact(in1 := "EngineRPM", in2 := "Settings".CATMinRPM)
      { S7_Templates := "time_type := Time" } #EngineFault_TON.TON(pt := "Settings".CATFaultTime, et =>)
      Coil( "EngineFault" )
   END_RUNG
   // the same network as SCL:
   #EngineFault_TON(IN := "StartCAT" AND ("EngineRPM" < "Settings".CATMinRPM), PT := "Settings".CATFaultTime);   // TON
   "EngineFault" := #EngineFault_TON.Q;
END_REGION
END_FUNCTION_BLOCK

FUNCTION_BLOCK "System_Enable"   // FB15, LAD
{ S7_Optimized_Access := 'TRUE' }
// Written BY Kristopher Gimenez January 26,2023
// This block is used to control enable the Pump and Fail safe valves based on HPU Startup.
// stored: AutoNumber false, MemoryReserve 100, SetENOAutomatically false
BEGIN

REGION Network 1: Enable System
   // Turn On Pump Enable and Fail save if Pumps have started or tried and are off ,with an elec HPU. 
   // Turn On Pump Enable and Fail Save if StartCAt
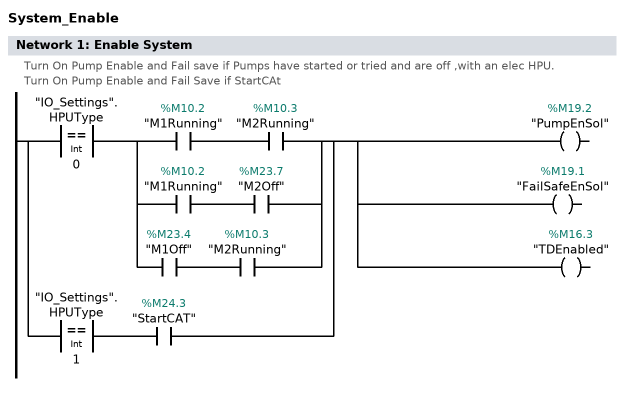
   RUNG wire#powerrail
      { S7_Templates := "SrcType := Int" } EQ_Contact(in1 := "IO_Settings".HPUType, in2 := 0)
      wire#w1
      Contact( "M1Running" )
      Contact( "M2Running" )
      wire#w2
      Coil( "PumpEnSol" )
   END_RUNG
   RUNG wire#w1
      Contact( "M1Running" )
      Contact( "M2Off" )
   END_RUNG wire#w2
   RUNG wire#w1
      Contact( "M1Off" )
      Contact( "M2Running" )
   END_RUNG wire#w2
   RUNG wire#powerrail
      { S7_Templates := "SrcType := Int" } EQ_Contact(in1 := "IO_Settings".HPUType, in2 := 1)
      Contact( "StartCAT" )
   END_RUNG wire#w2
   RUNG wire#w2
      Coil( "FailSafeEnSol" )
   END_RUNG
   RUNG wire#w2
      Coil( "TDEnabled" )
   END_RUNG
   // the same network as SCL:
   "PumpEnSol" := (("IO_Settings".HPUType = 0) AND (("M1Running" AND "M2Running") OR ("M1Running" AND "M2Off") OR ("M1Off" AND "M2Running"))) OR (("IO_Settings".HPUType = 1) AND "StartCAT");
   "FailSafeEnSol" := "PumpEnSol";
   "TDEnabled" := "PumpEnSol";
END_REGION
END_FUNCTION_BLOCK

FUNCTION_BLOCK "Aux_Functions"   // FB16, LAD
TITLE = Aux_Functions
{ S7_Optimized_Access := 'TRUE' }
// Written BY Kristopher Gimenez January 26,2023
// This block is used to control TD auxilarry functions
// stored: AutoNumber false, MemoryReserve 100, SetENOAutomatically false
   VAR
      PTO_Pulse { S7_SetPoint := 'True'} : TP_TIME;
      BUWOpenCLKTOffTime { S7_SetPoint := 'True'} : TP_TIME;
      BUWOpenCLKOnTime { S7_SetPoint := 'True'} : TP_TIME;
      BUWCloseHoldTOF { S7_SetPoint := 'True'} : TOF_TIME;
      MUDoneTP { S7_SetPoint := 'True'} : TP_TIME;
      BUWOpPulse { S7_SetPoint := 'True'} : TP_TIME;
      ElevCl_TON { S7_SetPoint := 'True'} : TON_TIME;
      ElevOpTime_TP { S7_SetPoint := 'True'} : TP_TIME;
      MSVOp_TON { S7_SetPoint := 'True'} : TON_TIME;
      MPRunning_TOF { S7_SetPoint := 'True'} : TOF_TIME;
      MSVCl_TON { S7_SetPoint := 'True'} : TON_TIME;
      BUWMainCl_Int { S7_SetPoint := 'True'} : Bool;
      TDModeMUTrig : Bool;
      TDModeBOTrig { ExternalAccessible := 'False'; ExternalVisible := 'False'; ExternalWritable := 'False'} : Bool;
      ElevOpOnTime : Bool;   // Bool that will be high for 8 seconds while elevator opens
      LinksDisable : Bool;   // Link Tilt Extend and Retract disabled
      ElevClDisable : Bool;   // Disable Close after output on for set time
      MSVClDisable { S7_SetPoint := 'True'} : Bool;   // MSV close disabled due to mud Pump running if high
      MSVOpDisable { S7_SetPoint := 'True'} : Bool;   // Disable after output on for set time
      ElevOpSwTrig : Bool;
      ElevCl_TON_1 { S7_SetPoint := 'True'} : TON_TIME;
      ElevCl_TON_5s { S7_SetPoint := 'True'} : TON_TIME;
   END_VAR
   // PTO_Pulse.PT := T#5s;
   VAR_TEMP   // added for the SCL form of the ladder/FBD networks
      _w1 : Bool;
      _w2 : Bool;
   END_VAR
BEGIN

REGION Network 1: PTO Pulse
   // When PTO is pressed there will be a 5 seconds pulse allowing operations.
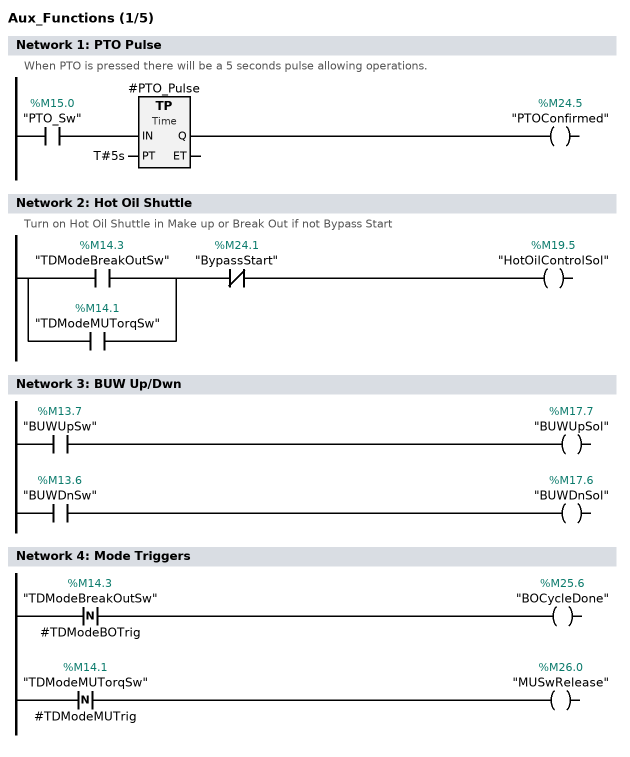
   RUNG wire#powerrail
      Contact( "PTO_Sw" )
      { S7_Templates := "time_type := Time" } #PTO_Pulse.TP(pt := T#5s, et =>)
      Coil( "PTOConfirmed" )
   END_RUNG
   // the same network as SCL:
   #PTO_Pulse(IN := "PTO_Sw", PT := T#5s);   // TP
   "PTOConfirmed" := #PTO_Pulse.Q;
END_REGION

REGION Network 2: Hot Oil Shuttle
   // Turn on Hot Oil Shuttle in Make up or Break Out if not Bypass Start
   RUNG wire#powerrail
      Contact( "TDModeBreakOutSw" )
      wire#w1
      I_Contact( "BypassStart" )
      Coil( "HotOilControlSol" )
   END_RUNG
   RUNG wire#powerrail
      Contact( "TDModeMUTorqSw" )
   END_RUNG wire#w1
   // the same network as SCL:
   "HotOilControlSol" := ("TDModeBreakOutSw" OR "TDModeMUTorqSw") AND NOT "BypassStart";
END_REGION

REGION Network 3: BUW Up/Dwn
   RUNG wire#powerrail
      Contact( "BUWUpSw" )
      Coil( "BUWUpSol" )
   END_RUNG
   RUNG wire#powerrail
      Contact( "BUWDnSw" )
      Coil( "BUWDnSol" )
   END_RUNG
   // the same network as SCL:
   "BUWUpSol" := "BUWUpSw";
   "BUWDnSol" := "BUWDnSw";
END_REGION

REGION Network 4: Mode Triggers
   RUNG wire#powerrail
      N_Contact(operand := "TDModeBreakOutSw", bit := #TDModeBOTrig)
      Coil( "BOCycleDone" )
   END_RUNG
   RUNG wire#powerrail
      N_Contact(operand := "TDModeMUTorqSw", bit := #TDModeMUTrig)
      Coil( "MUSwRelease" )
   END_RUNG
   // the same network as SCL:
   #_w1 := NOT "TDModeBreakOutSw" AND #TDModeBOTrig;   // falling edge of "TDModeBreakOutSw"
   #TDModeBOTrig := "TDModeBreakOutSw";
   "BOCycleDone" := #_w1;
   #_w2 := NOT "TDModeMUTorqSw" AND #TDModeMUTrig;   // falling edge of "TDModeMUTorqSw"
   #TDModeMUTrig := "TDModeMUTorqSw";
   "MUSwRelease" := #_w2;
END_REGION

REGION Network 5: BUW Close Latches
   // MaintContirm - PTO must be pressed before Quill Lock Switch Engage and rotary stopped- Set/Reset Maint
   // Hold Close Time set if TD Mode Sw is used while Auto Closing. Reset if not Auto Closing an all Sw off.
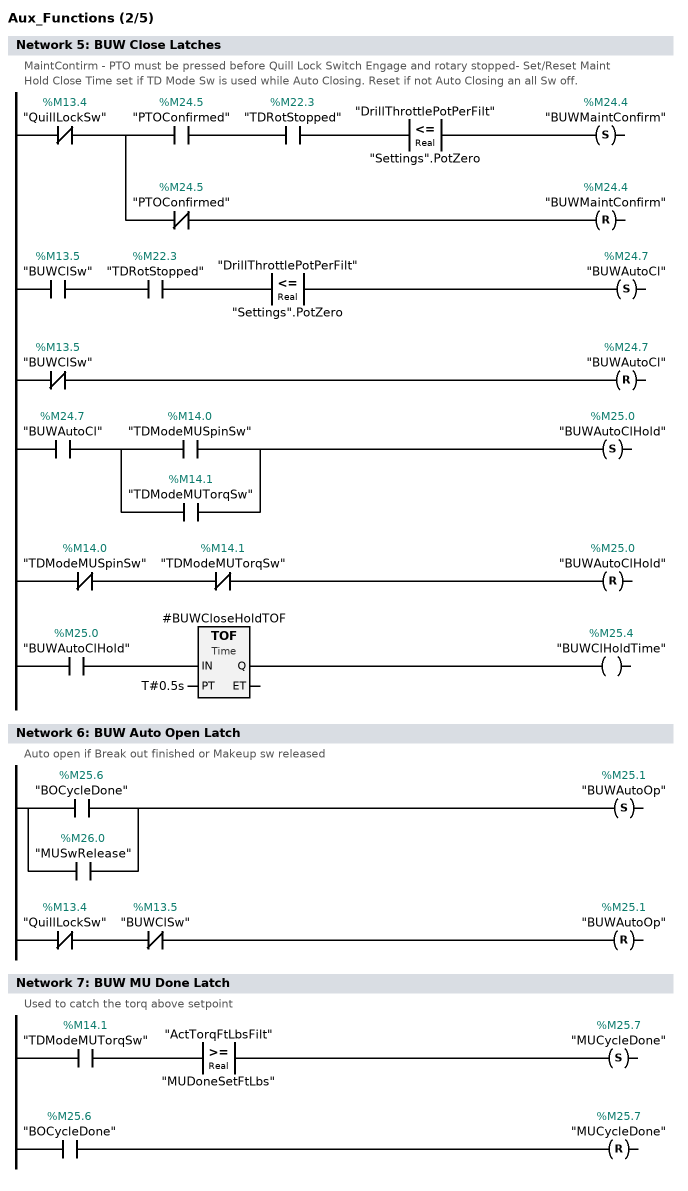
   RUNG wire#powerrail
      I_Contact( "QuillLockSw" )
      wire#w1
      Contact( "PTOConfirmed" )
      Contact( "TDRotStopped" )
      { S7_Templates := "SrcType := Real" } LE_Contact(in1 := "DrillThrottlePotPerFilt", in2 := "Settings".PotZero)
      S_Coil( "BUWMaintConfirm" )
   END_RUNG
   RUNG wire#w1
      I_Contact( "PTOConfirmed" )
      R_Coil( "BUWMaintConfirm" )
   END_RUNG
   RUNG wire#powerrail
      Contact( "BUWClSw" )
      Contact( "TDRotStopped" )
      { S7_Templates := "SrcType := Real" } LE_Contact(in1 := "DrillThrottlePotPerFilt", in2 := "Settings".PotZero)
      S_Coil( "BUWAutoCl" )
   END_RUNG
   RUNG wire#powerrail
      I_Contact( "BUWClSw" )
      R_Coil( "BUWAutoCl" )
   END_RUNG
   RUNG wire#powerrail
      Contact( "BUWAutoCl" )
      wire#w2
      Contact( "TDModeMUSpinSw" )
      wire#w3
      S_Coil( "BUWAutoClHold" )
   END_RUNG
   RUNG wire#w2
      Contact( "TDModeMUTorqSw" )
   END_RUNG wire#w3
   RUNG wire#powerrail
      I_Contact( "TDModeMUSpinSw" )
      I_Contact( "TDModeMUTorqSw" )
      R_Coil( "BUWAutoClHold" )
   END_RUNG
   RUNG wire#powerrail
      Contact( "BUWAutoClHold" )
      { S7_Templates := "time_type := Time" } #BUWCloseHoldTOF.TOF(pt := T#0.5s, et =>)
      Coil( "BUWClHoldTime" )
   END_RUNG
   // the same network as SCL:
   IF NOT "QuillLockSw" AND "PTOConfirmed" AND "TDRotStopped" AND ("DrillThrottlePotPerFilt" <= "Settings".PotZero) THEN
       "BUWMaintConfirm" := TRUE;
   END_IF;
   IF NOT "QuillLockSw" AND NOT "PTOConfirmed" THEN "BUWMaintConfirm" := FALSE; END_IF;
   IF "BUWClSw" AND "TDRotStopped" AND ("DrillThrottlePotPerFilt" <= "Settings".PotZero) THEN
       "BUWAutoCl" := TRUE;
   END_IF;
   IF NOT "BUWClSw" THEN "BUWAutoCl" := FALSE; END_IF;
   IF "BUWAutoCl" AND ("TDModeMUSpinSw" OR "TDModeMUTorqSw") THEN "BUWAutoClHold" := TRUE; END_IF;
   IF NOT "TDModeMUSpinSw" AND NOT "TDModeMUTorqSw" THEN "BUWAutoClHold" := FALSE; END_IF;
   #BUWCloseHoldTOF(IN := "BUWAutoClHold", PT := T#0.5s);   // TOF
   "BUWClHoldTime" := #BUWCloseHoldTOF.Q;
END_REGION

REGION Network 6: BUW Auto Open Latch
   // Auto open if Break out finished or Makeup sw released
   RUNG wire#powerrail
      Contact( "BOCycleDone" )
      wire#w1
      S_Coil( "BUWAutoOp" )
   END_RUNG
   RUNG wire#powerrail
      Contact( "MUSwRelease" )
   END_RUNG wire#w1
   RUNG wire#powerrail
      I_Contact( "QuillLockSw" )
      I_Contact( "BUWClSw" )
      R_Coil( "BUWAutoOp" )
   END_RUNG
   // the same network as SCL:
   IF "BOCycleDone" OR "MUSwRelease" THEN "BUWAutoOp" := TRUE; END_IF;
   IF NOT "QuillLockSw" AND NOT "BUWClSw" THEN "BUWAutoOp" := FALSE; END_IF;
END_REGION

REGION Network 7: BUW MU Done Latch
   // Used to catch the torq above setpoint
   RUNG wire#powerrail
      Contact( "TDModeMUTorqSw" )
      { S7_Templates := "SrcType := Real" } GE_Contact(in1 := "ActTorqFtLbsFilt", in2 := "MUDoneSetFtLbs")
      S_Coil( "MUCycleDone" )
   END_RUNG
   RUNG wire#powerrail
      Contact( "BOCycleDone" )
      R_Coil( "MUCycleDone" )
   END_RUNG
   // the same network as SCL:
   IF "TDModeMUTorqSw" AND ("ActTorqFtLbsFilt" >= "MUDoneSetFtLbs") THEN "MUCycleDone" := TRUE; END_IF;
   IF "BOCycleDone" THEN "MUCycleDone" := FALSE; END_IF;
END_REGION

REGION Network 8: BUW Sliding mode flag
   // Used to disabled Quill Lock if BO was last function performed. MU cycle must be completed to enable.
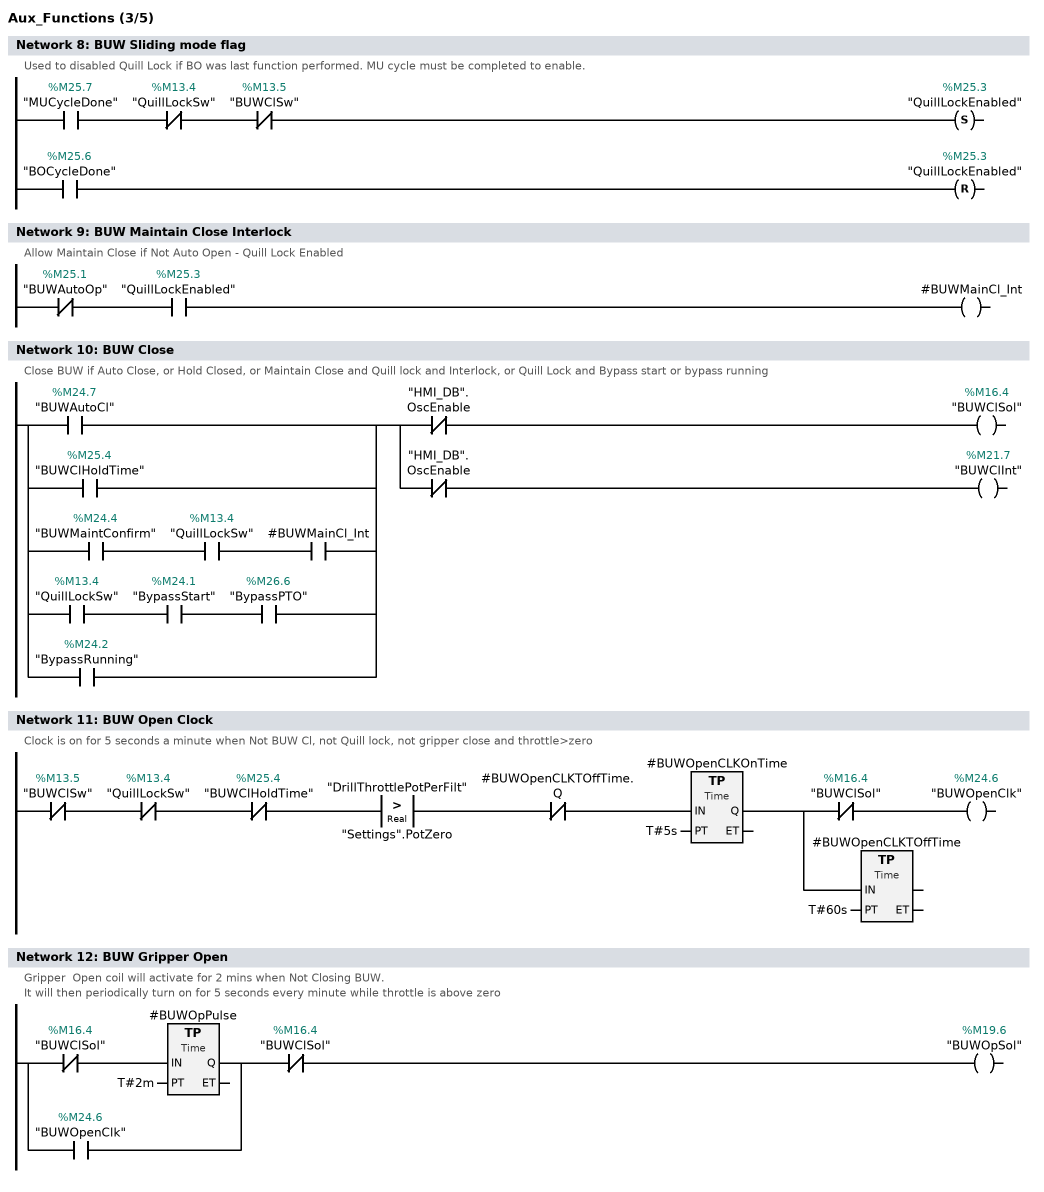
   RUNG wire#powerrail
      Contact( "MUCycleDone" )
      I_Contact( "QuillLockSw" )
      I_Contact( "BUWClSw" )
      S_Coil( "QuillLockEnabled" )
   END_RUNG
   RUNG wire#powerrail
      Contact( "BOCycleDone" )
      R_Coil( "QuillLockEnabled" )
   END_RUNG
   // the same network as SCL:
   IF "MUCycleDone" AND NOT "QuillLockSw" AND NOT "BUWClSw" THEN "QuillLockEnabled" := TRUE; END_IF;
   IF "BOCycleDone" THEN "QuillLockEnabled" := FALSE; END_IF;
END_REGION

REGION Network 9: BUW Maintain Close Interlock
   // Allow Maintain Close if Not Auto Open - Quill Lock Enabled
   RUNG wire#powerrail
      I_Contact( "BUWAutoOp" )
      Contact( "QuillLockEnabled" )
      Coil( #BUWMainCl_Int )
   END_RUNG
   // the same network as SCL:
   #BUWMainCl_Int := NOT "BUWAutoOp" AND "QuillLockEnabled";
END_REGION

REGION Network 10: BUW Close
   // Close BUW if Auto Close, or Hold Closed, or Maintain Close and Quill lock and Interlock, or Quill Lock and Bypass start or bypass running
   RUNG wire#powerrail
      Contact( "BUWAutoCl" )
      wire#w1
      I_Contact( "HMI_DB".OscEnable )
      Coil( "BUWClSol" )
   END_RUNG
   RUNG wire#powerrail
      Contact( "BUWClHoldTime" )
   END_RUNG wire#w1
   RUNG wire#powerrail
      Contact( "BUWMaintConfirm" )
      Contact( "QuillLockSw" )
      Contact( #BUWMainCl_Int )
   END_RUNG wire#w1
   RUNG wire#powerrail
      Contact( "QuillLockSw" )
      Contact( "BypassStart" )
      Contact( "BypassPTO" )
   END_RUNG wire#w1
   RUNG wire#powerrail
      Contact( "BypassRunning" )
   END_RUNG wire#w1
   RUNG wire#w1
      I_Contact( "HMI_DB".OscEnable )
      Coil( "BUWClInt" )
   END_RUNG
   // the same network as SCL:
   #_w1 := "BUWAutoCl" OR "BUWClHoldTime" OR ("BUWMaintConfirm" AND "QuillLockSw" AND #BUWMainCl_Int) OR ("QuillLockSw" AND "BypassStart" AND "BypassPTO") OR "BypassRunning";
   "BUWClSol" := #_w1 AND NOT "HMI_DB".OscEnable;
   "BUWClInt" := #_w1 AND NOT "HMI_DB".OscEnable;
END_REGION

REGION Network 11: BUW Open Clock
   // Clock is on for 5 seconds a minute when Not BUW Cl, not Quill lock, not gripper close and throttle>zero
   RUNG wire#powerrail
      I_Contact( "BUWClSw" )
      I_Contact( "QuillLockSw" )
      I_Contact( "BUWClHoldTime" )
      { S7_Templates := "SrcType := Real" } GT_Contact(in1 := "DrillThrottlePotPerFilt", in2 := "Settings".PotZero)
      I_Contact( #BUWOpenCLKTOffTime.Q )
      { S7_Templates := "time_type := Time" } #BUWOpenCLKOnTime.TP(pt := T#5s, et =>)
      wire#w1
      I_Contact( "BUWClSol" )
      Coil( "BUWOpenClk" )
   END_RUNG
   RUNG wire#w1
      { S7_Templates := "time_type := Time" } #BUWOpenCLKTOffTime.TP(pt := T#60s, et =>)
   END_RUNG
   // the same network as SCL:
   #BUWOpenCLKOnTime(IN := NOT "BUWClSw" AND NOT "QuillLockSw" AND NOT "BUWClHoldTime" AND ("DrillThrottlePotPerFilt" > "Settings".PotZero) AND NOT #BUWOpenCLKTOffTime.Q,   // TP
                     PT := T#5s);
   "BUWOpenClk" := #BUWOpenCLKOnTime.Q AND NOT "BUWClSol";
   #BUWOpenCLKTOffTime(IN := #BUWOpenCLKOnTime.Q, PT := T#60s);   // TP
END_REGION

REGION Network 12: BUW Gripper Open
   // Gripper  Open coil will activate for 2 mins when Not Closing BUW. 
   // It will then periodically turn on for 5 seconds every minute while throttle is above zero
   RUNG wire#powerrail
      I_Contact( "BUWClSol" )
      { S7_Templates := "time_type := Time" } #BUWOpPulse.TP(pt := T#2m, et =>)
      wire#w1
      I_Contact( "BUWClSol" )
      Coil( "BUWOpSol" )
   END_RUNG
   RUNG wire#powerrail
      Contact( "BUWOpenClk" )
   END_RUNG wire#w1
   // the same network as SCL:
   #BUWOpPulse(IN := NOT "BUWClSol", PT := T#2m);   // TP
   "BUWOpSol" := (#BUWOpPulse.Q OR "BUWOpenClk") AND NOT "BUWClSol";
END_REGION

REGION Network 13: Elevator Close
   // While SW held in close position hold output on for 10 s if no feedback,   or  hold for close position for 5s with feedback =1 (on)
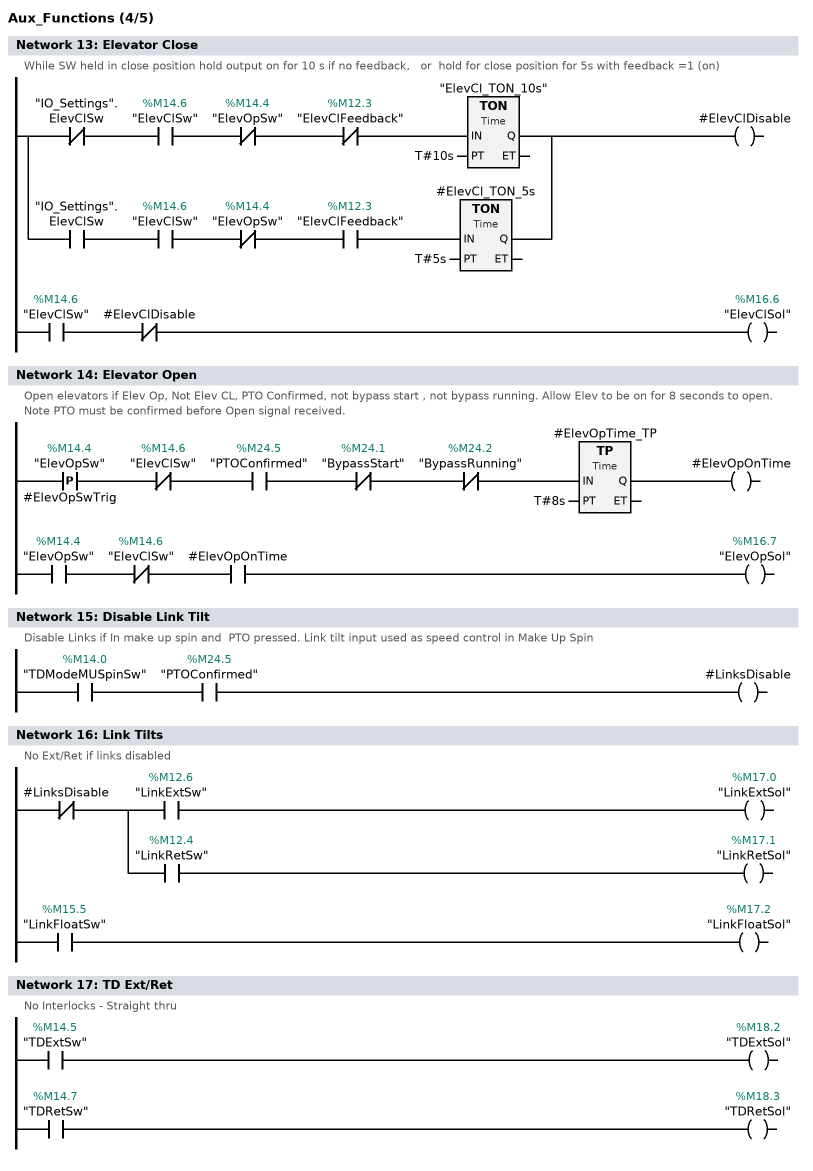
   RUNG wire#powerrail
      I_Contact( "IO_Settings".ElevClSw )
      Contact( "ElevClSw" )
      I_Contact( "ElevOpSw" )
      I_Contact( "ElevClFeedback" )
      { S7_Templates := "time_type := Time" } "ElevCl_TON_10s".TON(pt := T#10s, et =>)
      wire#w1
      Coil( #ElevClDisable )
   END_RUNG
   RUNG wire#powerrail
      Contact( "IO_Settings".ElevClSw )
      Contact( "ElevClSw" )
      I_Contact( "ElevOpSw" )
      Contact( "ElevClFeedback" )
      { S7_Templates := "time_type := Time" } #ElevCl_TON_5s.TON(pt := T#5s, et =>)
   END_RUNG wire#w1
   RUNG wire#powerrail
      Contact( "ElevClSw" )
      I_Contact( #ElevClDisable )
      Coil( "ElevClSol" )
   END_RUNG
   // the same network as SCL:
   "ElevCl_TON_10s".TON(IN := NOT "IO_Settings".ElevClSw AND "ElevClSw" AND NOT "ElevOpSw" AND NOT "ElevClFeedback",
                        PT := T#10s);
   #ElevCl_TON_5s(IN := "IO_Settings".ElevClSw AND "ElevClSw" AND NOT "ElevOpSw" AND "ElevClFeedback",   // TON
                  PT := T#5s);
   #ElevClDisable := "ElevCl_TON_10s".Q OR #ElevCl_TON_5s.Q;
   "ElevClSol" := "ElevClSw" AND NOT #ElevClDisable;
END_REGION

REGION Network 14: Elevator Open
   // Open elevators if Elev Op, Not Elev CL, PTO Confirmed, not bypass start , not bypass running. Allow Elev to be on for 8 seconds to open. Note PTO must be confirmed before Open signal received.
   RUNG wire#powerrail
      P_Contact(operand := "ElevOpSw", bit := #ElevOpSwTrig)
      I_Contact( "ElevClSw" )
      Contact( "PTOConfirmed" )
      I_Contact( "BypassStart" )
      I_Contact( "BypassRunning" )
      { S7_Templates := "time_type := Time" } #ElevOpTime_TP.TP(pt := T#8s, et =>)
      Coil( #ElevOpOnTime )
   END_RUNG
   RUNG wire#powerrail
      Contact( "ElevOpSw" )
      I_Contact( "ElevClSw" )
      Contact( #ElevOpOnTime )
      Coil( "ElevOpSol" )
   END_RUNG
   // the same network as SCL:
   #_w1 := "ElevOpSw" AND NOT #ElevOpSwTrig;   // rising edge of "ElevOpSw"
   #ElevOpSwTrig := "ElevOpSw";
   #ElevOpTime_TP(IN := #_w1 AND NOT "ElevClSw" AND "PTOConfirmed" AND NOT "BypassStart" AND NOT "BypassRunning",   // TP
                  PT := T#8s);
   #ElevOpOnTime := #ElevOpTime_TP.Q;
   "ElevOpSol" := "ElevOpSw" AND NOT "ElevClSw" AND #ElevOpOnTime;
END_REGION

REGION Network 15: Disable Link Tilt
   // Disable Links if In make up spin and  PTO pressed. Link tilt input used as speed control in Make Up Spin
   RUNG wire#powerrail
      Contact( "TDModeMUSpinSw" )
      Contact( "PTOConfirmed" )
      Coil( #LinksDisable )
   END_RUNG
   // the same network as SCL:
   #LinksDisable := "TDModeMUSpinSw" AND "PTOConfirmed";
END_REGION

REGION Network 16: Link Tilts
   // No Ext/Ret if links disabled
   RUNG wire#powerrail
      I_Contact( #LinksDisable )
      wire#w1
      Contact( "LinkExtSw" )
      Coil( "LinkExtSol" )
   END_RUNG
   RUNG wire#w1
      Contact( "LinkRetSw" )
      Coil( "LinkRetSol" )
   END_RUNG
   RUNG wire#powerrail
      Contact( "LinkFloatSw" )
      Coil( "LinkFloatSol" )
   END_RUNG
   // the same network as SCL:
   "LinkExtSol" := NOT #LinksDisable AND "LinkExtSw";
   "LinkRetSol" := NOT #LinksDisable AND "LinkRetSw";
   "LinkFloatSol" := "LinkFloatSw";
END_REGION

REGION Network 17: TD Ext/Ret
   // No Interlocks - Straight thru
   RUNG wire#powerrail
      Contact( "TDExtSw" )
      Coil( "TDExtSol" )
   END_RUNG
   RUNG wire#powerrail
      Contact( "TDRetSw" )
      Coil( "TDRetSol" )
   END_RUNG
   // the same network as SCL:
   "TDExtSol" := "TDExtSw";
   "TDRetSol" := "TDRetSw";
END_REGION

REGION Network 18: Handler FWD/Rev
   // No Interlocks - Straight thru
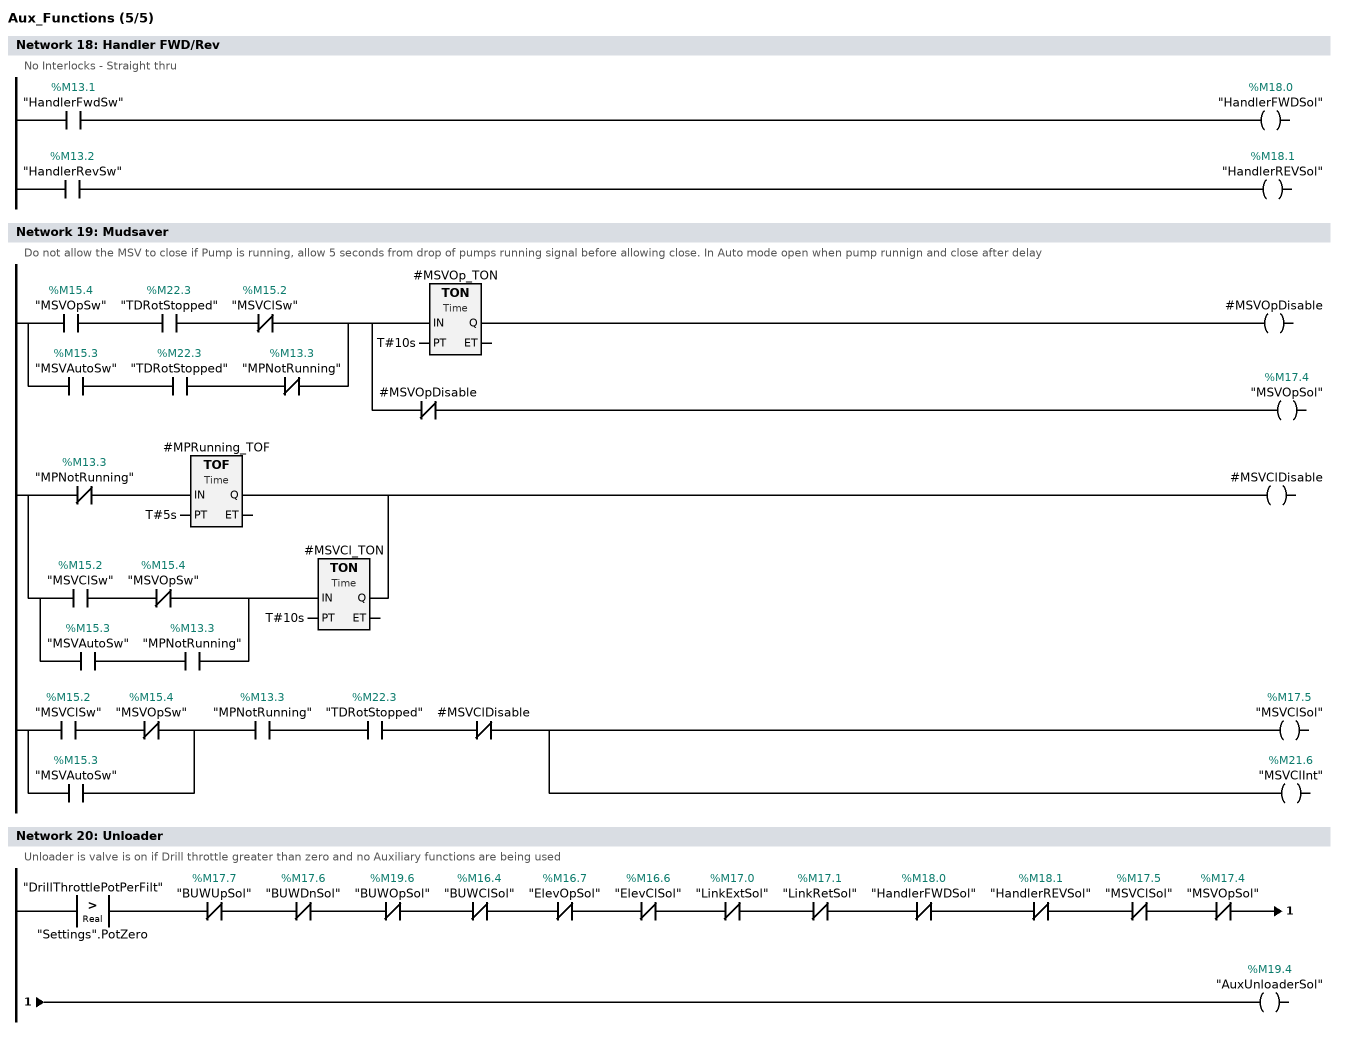
   RUNG wire#powerrail
      Contact( "HandlerFwdSw" )
      Coil( "HandlerFWDSol" )
   END_RUNG
   RUNG wire#powerrail
      Contact( "HandlerRevSw" )
      Coil( "HandlerREVSol" )
   END_RUNG
   // the same network as SCL:
   "HandlerFWDSol" := "HandlerFwdSw";
   "HandlerREVSol" := "HandlerRevSw";
END_REGION

REGION Network 19: Mudsaver
   // Do not allow the MSV to close if Pump is running, allow 5 seconds from drop of pumps running signal before allowing close. In Auto mode open when pump runnign and close after delay
   RUNG wire#powerrail
      Contact( "MSVOpSw" )
      Contact( "TDRotStopped" )
      I_Contact( "MSVClSw" )
      wire#w1
      { S7_Templates := "time_type := Time" } #MSVOp_TON.TON(pt := T#10s, et =>)
      Coil( #MSVOpDisable )
   END_RUNG
   RUNG wire#powerrail
      Contact( "MSVAutoSw" )
      Contact( "TDRotStopped" )
      I_Contact( "MPNotRunning" )
   END_RUNG wire#w1
   RUNG wire#w1
      I_Contact( #MSVOpDisable )
      Coil( "MSVOpSol" )
   END_RUNG
   RUNG wire#powerrail
      I_Contact( "MPNotRunning" )
      { S7_Templates := "time_type := Time" } #MPRunning_TOF.TOF(pt := T#5s, et =>)
      wire#w2
      Coil( #MSVClDisable )
   END_RUNG
   RUNG wire#powerrail
      Contact( "MSVClSw" )
      I_Contact( "MSVOpSw" )
      wire#w3
      { S7_Templates := "time_type := Time" } #MSVCl_TON.TON(pt := T#10s, et =>)
   END_RUNG wire#w2
   RUNG wire#powerrail
      Contact( "MSVAutoSw" )
      Contact( "MPNotRunning" )
   END_RUNG wire#w3
   RUNG wire#powerrail
      Contact( "MSVClSw" )
      I_Contact( "MSVOpSw" )
      wire#w4
      Contact( "MPNotRunning" )
      Contact( "TDRotStopped" )
      I_Contact( #MSVClDisable )
      wire#w5
      Coil( "MSVClSol" )
   END_RUNG
   RUNG wire#powerrail
      Contact( "MSVAutoSw" )
   END_RUNG wire#w4
   RUNG wire#w5
      Coil( "MSVClInt" )
   END_RUNG
   // the same network as SCL:
   #_w1 := ("MSVOpSw" AND "TDRotStopped" AND NOT "MSVClSw") OR ("MSVAutoSw" AND "TDRotStopped" AND NOT "MPNotRunning");
   #MSVOp_TON(IN := #_w1, PT := T#10s);   // TON
   #MSVOpDisable := #MSVOp_TON.Q;
   "MSVOpSol" := #_w1 AND NOT #MSVOpDisable;
   #MPRunning_TOF(IN := NOT "MPNotRunning", PT := T#5s);   // TOF
   #MSVCl_TON(IN := ("MSVClSw" AND NOT "MSVOpSw") OR ("MSVAutoSw" AND "MPNotRunning"), PT := T#10s);   // TON
   #MSVClDisable := #MPRunning_TOF.Q OR #MSVCl_TON.Q;
   "MSVClSol" := (("MSVClSw" AND NOT "MSVOpSw") OR "MSVAutoSw") AND "MPNotRunning" AND "TDRotStopped" AND NOT #MSVClDisable;
   "MSVClInt" := "MSVClSol";
END_REGION

REGION Network 20: Unloader
   // Unloader is valve is on if Drill throttle greater than zero and no Auxiliary functions are being used
   RUNG wire#powerrail
      { S7_Templates := "SrcType := Real" } GT_Contact(in1 := "DrillThrottlePotPerFilt", in2 := "Settings".PotZero)
      I_Contact( "BUWUpSol" )
      I_Contact( "BUWDnSol" )
      I_Contact( "BUWOpSol" )
      I_Contact( "BUWClSol" )
      I_Contact( "ElevOpSol" )
      I_Contact( "ElevClSol" )
      I_Contact( "LinkExtSol" )
      I_Contact( "LinkRetSol" )
      I_Contact( "HandlerFWDSol" )
      I_Contact( "HandlerREVSol" )
      I_Contact( "MSVClSol" )
      I_Contact( "MSVOpSol" )
      Coil( "AuxUnloaderSol" )
   END_RUNG
   // the same network as SCL:
   "AuxUnloaderSol" := ("DrillThrottlePotPerFilt" > "Settings".PotZero) AND NOT "BUWUpSol" AND NOT "BUWDnSol" AND NOT "BUWOpSol" AND NOT "BUWClSol" AND NOT "ElevOpSol" AND NOT "ElevClSol" AND NOT "LinkExtSol" AND NOT "LinkRetSol" AND NOT "HandlerFWDSol" AND NOT "HandlerREVSol" AND NOT "MSVClSol" AND NOT "MSVOpSol";
END_REGION
END_FUNCTION_BLOCK

FUNCTION_BLOCK "TD_Control"   // FB19, LAD
TITLE = TD_Control
{ S7_Optimized_Access := 'TRUE' }
// Written BY Kristopher Gimenez Feb1,2023
// This block is used to control the TD control mode, pump outputs and HSLT/LSHT shifting
// stored: AutoNumber false, MemoryReserve 100, SetENOAutomatically false
   VAR
      AllowShift : Bool;   // Allow speed change
      TD_Mode : Int;   // TD Mode, 0=Drill, 1=DrillRev, 2=MU-S, 3=MU-T, 4= BO, 5 OSC, 6 Bypass
      HSLTShift_TP { S7_SetPoint := 'True'} : TP_TIME;
      LSHTShift_TP { S7_SetPoint := 'True'} : TP_TIME;
      MUSpinComplete : Bool;   // Set once MU spin torq above setpoint
      TDP1FwdSetmA : Real;
      TDP2FwdSetmA : Real;
      TDP1RevSetmA : Real;
      TDP2RevSetmA : Real;
      TorqSetmA : Real;
      TDP1FwdEn : Bool;
      TDP2FwdEn : Bool;
      TDP1RevEn : Bool;
      TDP2RevEn : Bool;
      TorqEn : Bool;
      BypassDelay_TON { S7_SetPoint := 'True'} : TON_TIME;
      BypassRunning_TOF { S7_SetPoint := 'True'} : TOF_TIME;
      HSLT_Sol_Last { S7_SetPoint := 'True'} : Bool;
      LSHT_Sol_Last : Bool;
      AllowRev : Bool;   // Latch that will allow Drill rev if rotary has stopped
      SpeedLimiting : Bool;
      SpeedLimitmAOut : Real;
      SpeedLimitingTrig : Bool;   // Positive Trigger Last cycle value
      MUTorqStart : Bool;
      BOStart : Bool;
      OscStart : Bool;
      MUTorqStart_Trig : Bool;
      BOStart_Trig : Bool;
      OscStart_Trig : Bool;
      SpeedLimit_SlewDec { S7_SetPoint := 'True'} : "SlewDec";
      SpeedLimit_SlewInc { S7_SetPoint := 'True'} : "SlewInc";
      HiTempShutDown_TON { S7_SetPoint := 'True'} : TON_TIME;
   END_VAR
   VAR_TEMP
      FlowmAOutTemp : Real;
      TorqmAOutTemp : Real;
      TorqPSITemp : Real;
      TorquePSI : Real;
      tempReal : Real;
   END_VAR
   VAR CONSTANT
      Disabled : Int := 0;   // TD Mode State Machine
      Drill : Int := 1;   // TD Mode State Machine
      DrillReverse : Int := 2;   // TD Mode State Machine
      MUSpin : Int := 3;   // TD Mode State Machine
      MUTorq : Int := 4;   // TD Mode State Machine
      BO : Int := 5;   // TD Mode State Machine
      Oscillate : Int := 6;   // TD Mode State Machine
      Bypass : Int := 7;   // TD Mode State Machine
   END_VAR
   VAR_TEMP   // added for the SCL form of the ladder/FBD networks
      _w1 : Bool;
      _w2 : Bool;
      _w3 : Bool;
      _w4 : Bool;
   END_VAR
BEGIN

REGION Network 1: Control Mode
   // Determine Control Mode based on Console Inputs and interlocks.
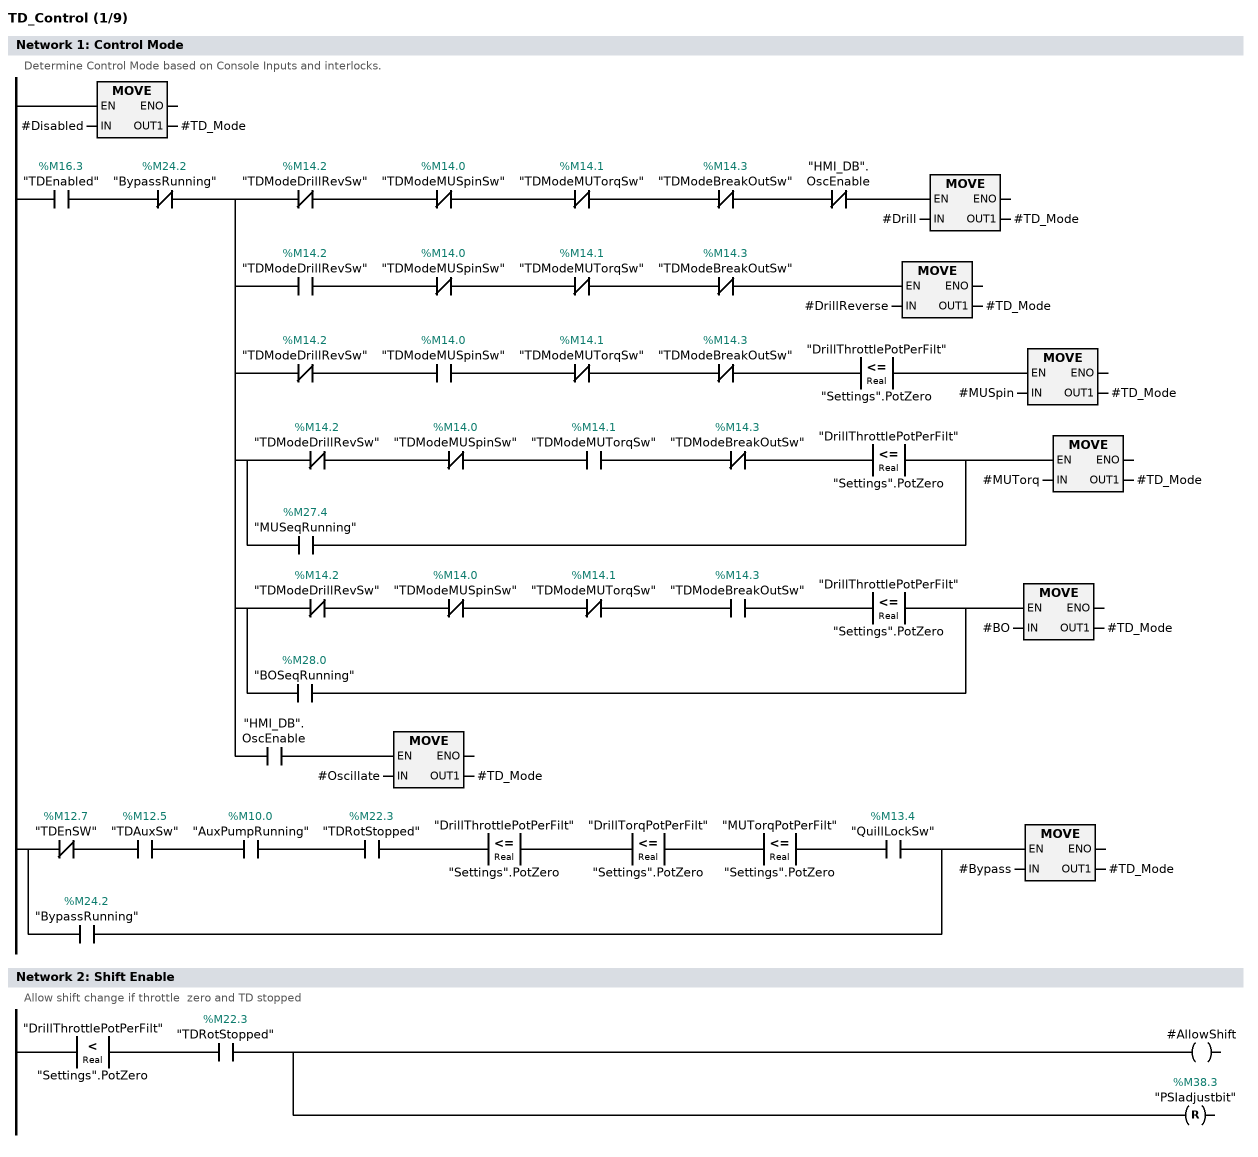
   RUNG wire#powerrail
      Move(in := #Disabled, out1 => #TD_Mode)
   END_RUNG
   RUNG wire#powerrail
      Contact( "TDEnabled" )
      I_Contact( "BypassRunning" )
      wire#w1
      I_Contact( "TDModeDrillRevSw" )
      I_Contact( "TDModeMUSpinSw" )
      I_Contact( "TDModeMUTorqSw" )
      I_Contact( "TDModeBreakOutSw" )
      I_Contact( "HMI_DB".OscEnable )
      Move(in := #Drill, out1 => #TD_Mode)
   END_RUNG
   RUNG wire#w1
      Contact( "TDModeDrillRevSw" )
      I_Contact( "TDModeMUSpinSw" )
      I_Contact( "TDModeMUTorqSw" )
      I_Contact( "TDModeBreakOutSw" )
      Move(in := #DrillReverse, out1 => #TD_Mode)
   END_RUNG
   RUNG wire#w1
      I_Contact( "TDModeDrillRevSw" )
      Contact( "TDModeMUSpinSw" )
      I_Contact( "TDModeMUTorqSw" )
      I_Contact( "TDModeBreakOutSw" )
      { S7_Templates := "SrcType := Real" } LE_Contact(in1 := "DrillThrottlePotPerFilt", in2 := "Settings".PotZero)
      Move(in := #MUSpin, out1 => #TD_Mode)
   END_RUNG
   RUNG wire#w1
      I_Contact( "TDModeDrillRevSw" )
      I_Contact( "TDModeMUSpinSw" )
      Contact( "TDModeMUTorqSw" )
      I_Contact( "TDModeBreakOutSw" )
      { S7_Templates := "SrcType := Real" } LE_Contact(in1 := "DrillThrottlePotPerFilt", in2 := "Settings".PotZero)
      wire#w2
      Move(in := #MUTorq, out1 => #TD_Mode)
   END_RUNG
   RUNG wire#w1
      Contact( "MUSeqRunning" )
   END_RUNG wire#w2
   RUNG wire#w1
      I_Contact( "TDModeDrillRevSw" )
      I_Contact( "TDModeMUSpinSw" )
      I_Contact( "TDModeMUTorqSw" )
      Contact( "TDModeBreakOutSw" )
      { S7_Templates := "SrcType := Real" } LE_Contact(in1 := "DrillThrottlePotPerFilt", in2 := "Settings".PotZero)
      wire#w3
      Move(in := #BO, out1 => #TD_Mode)
   END_RUNG
   RUNG wire#w1
      Contact( "BOSeqRunning" )
   END_RUNG wire#w3
   RUNG wire#w1
      Contact( "HMI_DB".OscEnable )
      Move(in := #Oscillate, out1 => #TD_Mode)
   END_RUNG
   RUNG wire#powerrail
      I_Contact( "TDEnSW" )
      Contact( "TDAuxSw" )
      Contact( "AuxPumpRunning" )
      Contact( "TDRotStopped" )
      { S7_Templates := "SrcType := Real" } LE_Contact(in1 := "DrillThrottlePotPerFilt", in2 := "Settings".PotZero)
      { S7_Templates := "SrcType := Real" } LE_Contact(in1 := "DrillTorqPotPerFilt", in2 := "Settings".PotZero)
      { S7_Templates := "SrcType := Real" } LE_Contact(in1 := "MUTorqPotPerFilt", in2 := "Settings".PotZero)
      Contact( "QuillLockSw" )
      wire#w4
      Move(in := #Bypass, out1 => #TD_Mode)
   END_RUNG
   RUNG wire#powerrail
      Contact( "BypassRunning" )
   END_RUNG wire#w4
   // the same network as SCL:
   #TD_Mode := #Disabled;
   #_w1 := "TDEnabled" AND NOT "BypassRunning";
   IF #_w1 AND NOT "TDModeDrillRevSw" AND NOT "TDModeMUSpinSw" AND NOT "TDModeMUTorqSw" AND NOT "TDModeBreakOutSw" AND NOT "HMI_DB".OscEnable THEN
       #TD_Mode := #Drill;
   END_IF;
   IF #_w1 AND "TDModeDrillRevSw" AND NOT "TDModeMUSpinSw" AND NOT "TDModeMUTorqSw" AND NOT "TDModeBreakOutSw" THEN
       #TD_Mode := #DrillReverse;
   END_IF;
   IF #_w1 AND NOT "TDModeDrillRevSw" AND "TDModeMUSpinSw" AND NOT "TDModeMUTorqSw" AND NOT "TDModeBreakOutSw" AND ("DrillThrottlePotPerFilt" <= "Settings".PotZero) THEN
       #TD_Mode := #MUSpin;
   END_IF;
   IF #_w1 AND ((NOT "TDModeDrillRevSw" AND NOT "TDModeMUSpinSw" AND "TDModeMUTorqSw" AND NOT "TDModeBreakOutSw" AND ("DrillThrottlePotPerFilt" <= "Settings".PotZero)) OR "MUSeqRunning") THEN
       #TD_Mode := #MUTorq;
   END_IF;
   IF #_w1 AND ((NOT "TDModeDrillRevSw" AND NOT "TDModeMUSpinSw" AND NOT "TDModeMUTorqSw" AND "TDModeBreakOutSw" AND ("DrillThrottlePotPerFilt" <= "Settings".PotZero)) OR "BOSeqRunning") THEN
       #TD_Mode := #BO;
   END_IF;
   IF #_w1 AND "HMI_DB".OscEnable THEN #TD_Mode := #Oscillate; END_IF;
   IF (NOT "TDEnSW" AND "TDAuxSw" AND "AuxPumpRunning" AND "TDRotStopped" AND ("DrillThrottlePotPerFilt" <= "Settings".PotZero) AND ("DrillTorqPotPerFilt" <= "Settings".PotZero) AND ("MUTorqPotPerFilt" <= "Settings".PotZero) AND "QuillLockSw") OR "BypassRunning" THEN
       #TD_Mode := #Bypass;
   END_IF;
END_REGION

REGION Network 2: Shift Enable
   // Allow shift change if throttle  zero and TD stopped
   RUNG wire#powerrail
      { S7_Templates := "SrcType := Real" } LT_Contact(in1 := "DrillThrottlePotPerFilt", in2 := "Settings".PotZero)
      Contact( "TDRotStopped" )
      wire#w1
      Coil( #AllowShift )
   END_RUNG
   RUNG wire#w1
      R_Coil( "PSIadjustbit" )
   END_RUNG
   // the same network as SCL:
   #AllowShift := ("DrillThrottlePotPerFilt" < "Settings".PotZero) AND "TDRotStopped";
   IF #AllowShift THEN "PSIadjustbit" := FALSE; END_IF;
END_REGION

REGION Network 3: HSLT/LSHT
   // Allow Shifting.  
   // Bypass in HSLT.  
   // MU modes, BO and Osc in LSHT. 
   // Drill modes follow console input
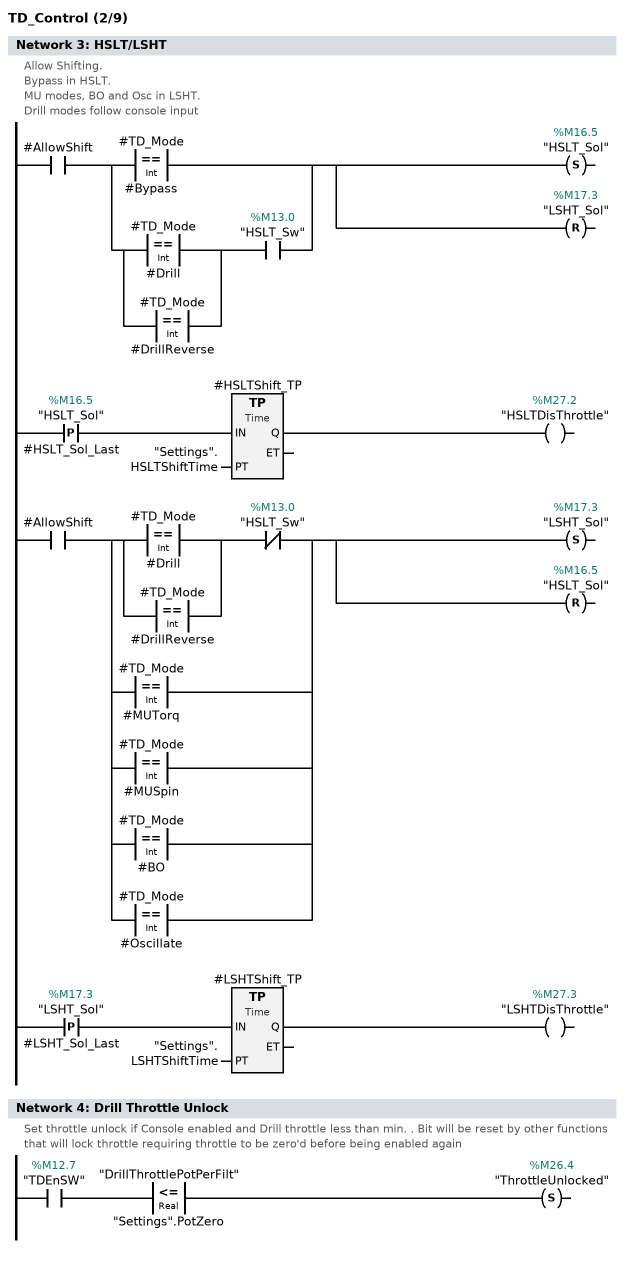
   RUNG wire#powerrail
      Contact( #AllowShift )
      wire#w1
      { S7_Templates := "SrcType := Int" } EQ_Contact(in1 := #TD_Mode, in2 := #Bypass)
      wire#w2
      S_Coil( "HSLT_Sol" )
   END_RUNG
   RUNG wire#w1
      { S7_Templates := "SrcType := Int" } EQ_Contact(in1 := #TD_Mode, in2 := #Drill)
      wire#w3
      Contact( "HSLT_Sw" )
   END_RUNG wire#w2
   RUNG wire#w1
      { S7_Templates := "SrcType := Int" } EQ_Contact(in1 := #TD_Mode, in2 := #DrillReverse)
   END_RUNG wire#w3
   RUNG wire#w2
      R_Coil( "LSHT_Sol" )
   END_RUNG
   RUNG wire#powerrail
      P_Contact(operand := "HSLT_Sol", bit := #HSLT_Sol_Last)
      { S7_Templates := "time_type := Time" } #HSLTShift_TP.TP(pt := "Settings".HSLTShiftTime, et =>)
      Coil( "HSLTDisThrottle" )
   END_RUNG
   RUNG wire#powerrail
      Contact( #AllowShift )
      wire#w4
      { S7_Templates := "SrcType := Int" } EQ_Contact(in1 := #TD_Mode, in2 := #Drill)
      wire#w5
      I_Contact( "HSLT_Sw" )
      wire#w6
      S_Coil( "LSHT_Sol" )
   END_RUNG
   RUNG wire#w4
      { S7_Templates := "SrcType := Int" } EQ_Contact(in1 := #TD_Mode, in2 := #DrillReverse)
   END_RUNG wire#w5
   RUNG wire#w4
      { S7_Templates := "SrcType := Int" } EQ_Contact(in1 := #TD_Mode, in2 := #MUTorq)
   END_RUNG wire#w6
   RUNG wire#w4
      { S7_Templates := "SrcType := Int" } EQ_Contact(in1 := #TD_Mode, in2 := #MUSpin)
   END_RUNG wire#w6
   RUNG wire#w4
      { S7_Templates := "SrcType := Int" } EQ_Contact(in1 := #TD_Mode, in2 := #BO)
   END_RUNG wire#w6
   RUNG wire#w4
      { S7_Templates := "SrcType := Int" } EQ_Contact(in1 := #TD_Mode, in2 := #Oscillate)
   END_RUNG wire#w6
   RUNG wire#w6
      R_Coil( "HSLT_Sol" )
   END_RUNG
   RUNG wire#powerrail
      P_Contact(operand := "LSHT_Sol", bit := #LSHT_Sol_Last)
      { S7_Templates := "time_type := Time" } #LSHTShift_TP.TP(pt := "Settings".LSHTShiftTime, et =>)
      Coil( "LSHTDisThrottle" )
   END_RUNG
   // the same network as SCL:
   IF #AllowShift AND ((#TD_Mode = #Bypass) OR (((#TD_Mode = #Drill) OR (#TD_Mode = #DrillReverse)) AND "HSLT_Sw")) THEN
       "HSLT_Sol" := TRUE;
       "LSHT_Sol" := FALSE;
   END_IF;
   #_w1 := "HSLT_Sol" AND NOT #HSLT_Sol_Last;   // rising edge of "HSLT_Sol"
   #HSLT_Sol_Last := "HSLT_Sol";
   #HSLTShift_TP(IN := #_w1, PT := "Settings".HSLTShiftTime);   // TP
   "HSLTDisThrottle" := #HSLTShift_TP.Q;
   IF #AllowShift AND ((((#TD_Mode = #Drill) OR (#TD_Mode = #DrillReverse)) AND NOT "HSLT_Sw") OR (#TD_Mode = #MUTorq) OR (#TD_Mode = #MUSpin) OR (#TD_Mode = #BO) OR (#TD_Mode = #Oscillate)) THEN
       "LSHT_Sol" := TRUE;
       "HSLT_Sol" := FALSE;
   END_IF;
   #_w2 := "LSHT_Sol" AND NOT #LSHT_Sol_Last;   // rising edge of "LSHT_Sol"
   #LSHT_Sol_Last := "LSHT_Sol";
   #LSHTShift_TP(IN := #_w2, PT := "Settings".LSHTShiftTime);   // TP
   "LSHTDisThrottle" := #LSHTShift_TP.Q;
END_REGION

REGION Network 4: Drill Throttle Unlock
   // Set throttle unlock if Console enabled and Drill throttle less than min. . Bit will be reset by other functions that will lock throttle requiring throttle to be zero'd before being enabled again
   RUNG wire#powerrail
      Contact( "TDEnSW" )
      { S7_Templates := "SrcType := Real" } LE_Contact(in1 := "DrillThrottlePotPerFilt", in2 := "Settings".PotZero)
      S_Coil( "ThrottleUnlocked" )
   END_RUNG
   // the same network as SCL:
   IF "TDEnSW" AND ("DrillThrottlePotPerFilt" <= "Settings".PotZero) THEN "ThrottleUnlocked" := TRUE; END_IF;
END_REGION

REGION Network 5: Drill Throttle Disable
   // Disable throttle if Bypass, Throttle disabled due to shift, or Flush fault or if throttle not unlocked
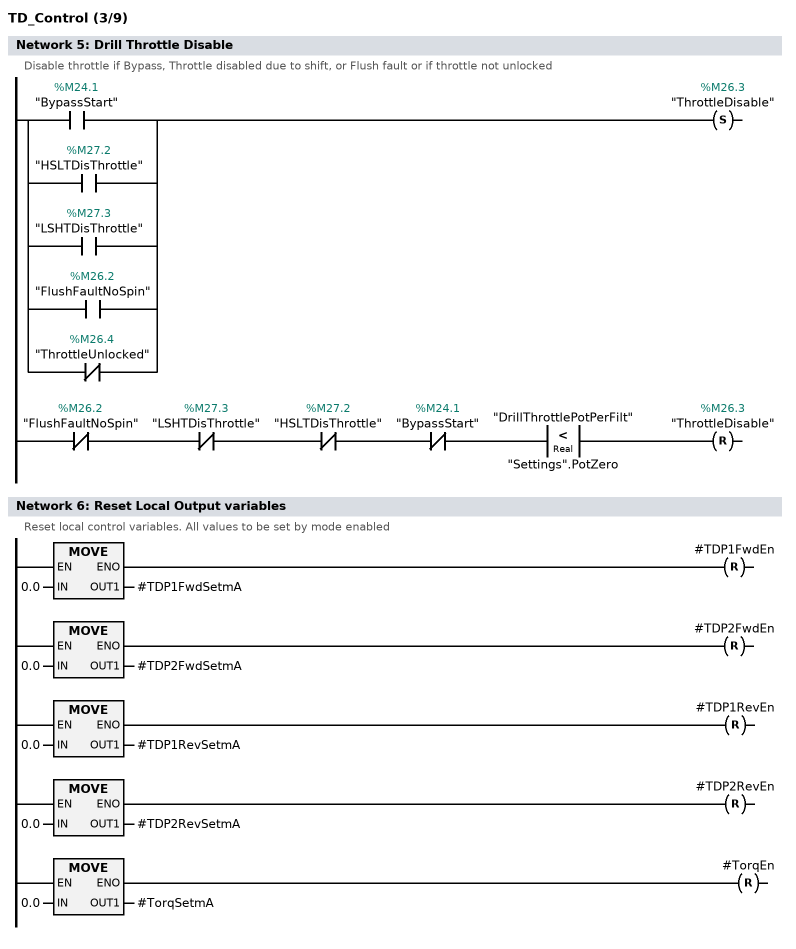
   RUNG wire#powerrail
      Contact( "BypassStart" )
      wire#w1
      S_Coil( "ThrottleDisable" )
   END_RUNG
   RUNG wire#powerrail
      Contact( "HSLTDisThrottle" )
   END_RUNG wire#w1
   RUNG wire#powerrail
      Contact( "LSHTDisThrottle" )
   END_RUNG wire#w1
   RUNG wire#powerrail
      Contact( "FlushFaultNoSpin" )
   END_RUNG wire#w1
   RUNG wire#powerrail
      I_Contact( "ThrottleUnlocked" )
   END_RUNG wire#w1
   RUNG wire#powerrail
      I_Contact( "FlushFaultNoSpin" )
      I_Contact( "LSHTDisThrottle" )
      I_Contact( "HSLTDisThrottle" )
      I_Contact( "BypassStart" )
      { S7_Templates := "SrcType := Real" } LT_Contact(in1 := "DrillThrottlePotPerFilt", in2 := "Settings".PotZero)
      R_Coil( "ThrottleDisable" )
   END_RUNG
   // the same network as SCL:
   IF "BypassStart" OR "HSLTDisThrottle" OR "LSHTDisThrottle" OR "FlushFaultNoSpin" OR NOT "ThrottleUnlocked" THEN
       "ThrottleDisable" := TRUE;
   END_IF;
   IF NOT "FlushFaultNoSpin" AND NOT "LSHTDisThrottle" AND NOT "HSLTDisThrottle" AND NOT "BypassStart" AND ("DrillThrottlePotPerFilt" < "Settings".PotZero) THEN
       "ThrottleDisable" := FALSE;
   END_IF;
END_REGION

REGION Network 6: Reset Local Output variables
   // Reset local control variables. All values to be set by mode enabled
   RUNG wire#powerrail
      Move(in := 0.0, out1 => #TDP1FwdSetmA)
      R_Coil( #TDP1FwdEn )
   END_RUNG
   RUNG wire#powerrail
      Move(in := 0.0, out1 => #TDP2FwdSetmA)
      R_Coil( #TDP2FwdEn )
   END_RUNG
   RUNG wire#powerrail
      Move(in := 0.0, out1 => #TDP1RevSetmA)
      R_Coil( #TDP1RevEn )
   END_RUNG
   RUNG wire#powerrail
      Move(in := 0.0, out1 => #TDP2RevSetmA)
      R_Coil( #TDP2RevEn )
   END_RUNG
   RUNG wire#powerrail
      Move(in := 0.0, out1 => #TorqSetmA)
      R_Coil( #TorqEn )
   END_RUNG
   // the same network as SCL:
   #TDP1FwdSetmA := 0.0;
   #TDP1FwdEn := FALSE;
   #TDP2FwdSetmA := 0.0;
   #TDP2FwdEn := FALSE;
   #TDP1RevSetmA := 0.0;
   #TDP1RevEn := FALSE;
   #TDP2RevSetmA := 0.0;
   #TDP2RevEn := FALSE;
   #TorqSetmA := 0.0;
   #TorqEn := FALSE;
END_REGION

REGION Network 7: Drill
   // In Drill Mode,
   // Torq Pot command is always sent to Torq valve. 
   // Throttle command to both Forward pumps if throttle not disabled and Throttle Above setpoint.
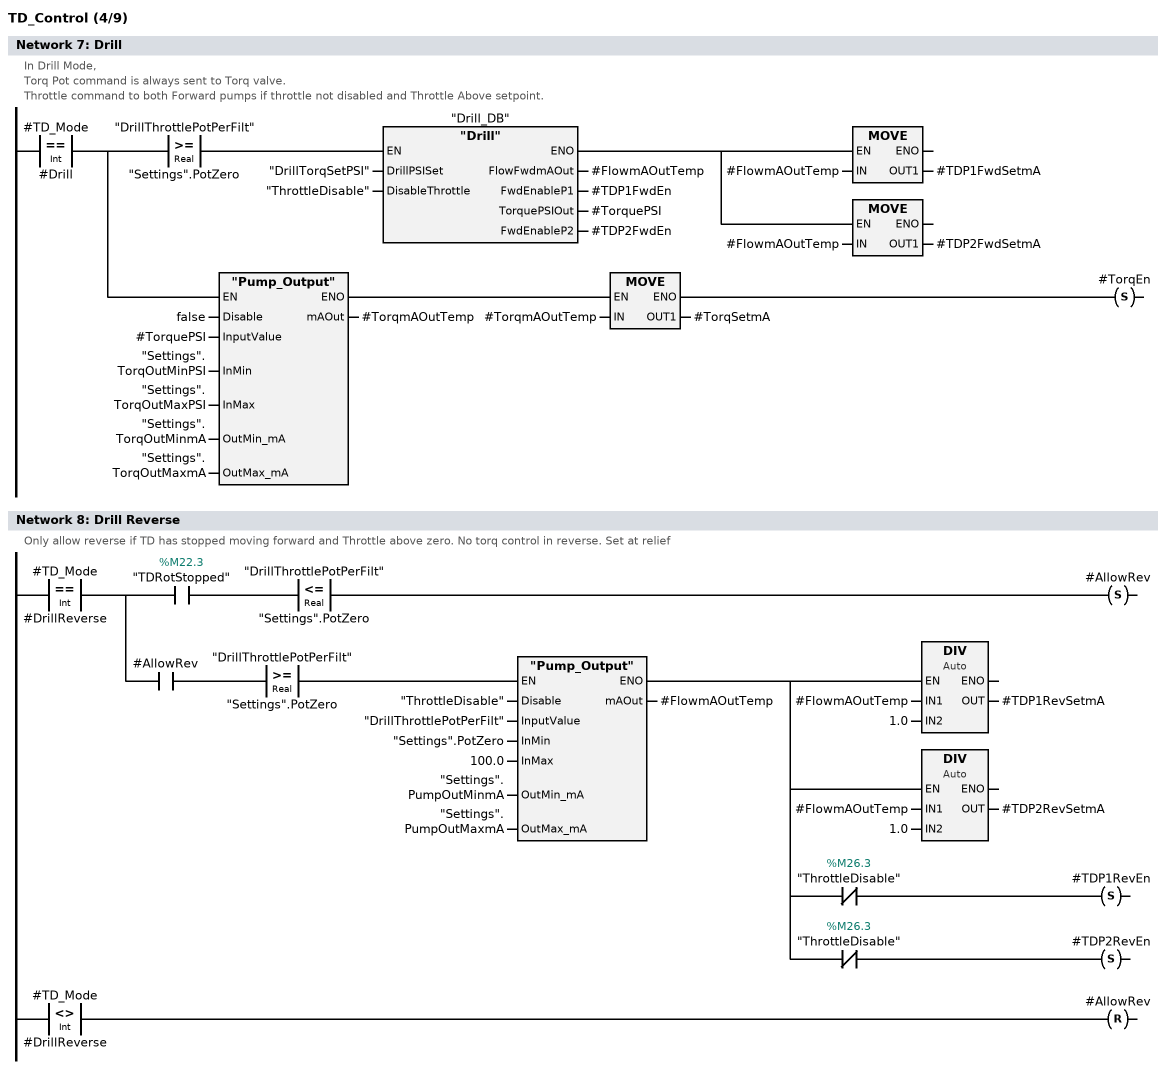
   RUNG wire#powerrail
      { S7_Templates := "SrcType := Int" } EQ_Contact(in1 := #TD_Mode, in2 := #Drill)
      wire#w1
      { S7_Templates := "SrcType := Real" } GE_Contact(in1 := "DrillThrottlePotPerFilt", in2 := "Settings".PotZero)
      "Drill_DB"(DrillPSISet := "DrillTorqSetPSI", DisableThrottle := "ThrottleDisable", FlowFwdmAOut => #FlowmAOutTemp, FwdEnableP1 => #TDP1FwdEn, TorquePSIOut => #TorquePSI, FwdEnableP2 => #TDP2FwdEn)
      wire#w2
      Move(in := #FlowmAOutTemp, out1 => #TDP1FwdSetmA)
   END_RUNG
   RUNG wire#w2
      Move(in := #FlowmAOutTemp, out1 => #TDP2FwdSetmA)
   END_RUNG
   RUNG wire#w1
      "Pump_Output"(Disable := false, InputValue := #TorquePSI, InMin := "Settings".TorqOutMinPSI, InMax := "Settings".TorqOutMaxPSI, OutMin_mA := "Settings".TorqOutMinmA, OutMax_mA := "Settings".TorqOutMaxmA, mAOut => #TorqmAOutTemp)
      Move(in := #TorqmAOutTemp, out1 => #TorqSetmA)
      S_Coil( #TorqEn )
   END_RUNG
   // the same network as SCL:
   #_w1 := #TD_Mode = #Drill;
   "Drill_DB"(EN := #_w1 AND ("DrillThrottlePotPerFilt" >= "Settings".PotZero),   // "Drill"
              DrillPSISet := "DrillTorqSetPSI",
              DisableThrottle := "ThrottleDisable",
              FlowFwdmAOut => #FlowmAOutTemp,
              FwdEnableP1 => #TDP1FwdEn,
              TorquePSIOut => #TorquePSI,
              FwdEnableP2 => #TDP2FwdEn,
              ENO => #_w2);
   IF #_w2 THEN
       #TDP1FwdSetmA := #FlowmAOutTemp;
       #TDP2FwdSetmA := #FlowmAOutTemp;
   END_IF;
   "Pump_Output"(EN := #_w1,
                 Disable := false,
                 InputValue := #TorquePSI,
                 InMin := "Settings".TorqOutMinPSI,
                 InMax := "Settings".TorqOutMaxPSI,
                 OutMin_mA := "Settings".TorqOutMinmA,
                 OutMax_mA := "Settings".TorqOutMaxmA,
                 mAOut => #TorqmAOutTemp,
                 ENO => #_w3);
   IF #_w3 THEN
       #TorqSetmA := #TorqmAOutTemp;
       #TorqEn := TRUE;
   END_IF;
END_REGION

REGION Network 8: Drill Reverse
   // Only allow reverse if TD has stopped moving forward and Throttle above zero. No torq control in reverse. Set at relief
   RUNG wire#powerrail
      { S7_Templates := "SrcType := Int" } EQ_Contact(in1 := #TD_Mode, in2 := #DrillReverse)
      wire#w1
      Contact( "TDRotStopped" )
      { S7_Templates := "SrcType := Real" } LE_Contact(in1 := "DrillThrottlePotPerFilt", in2 := "Settings".PotZero)
      S_Coil( #AllowRev )
   END_RUNG
   RUNG wire#w1
      Contact( #AllowRev )
      { S7_Templates := "SrcType := Real" } GE_Contact(in1 := "DrillThrottlePotPerFilt", in2 := "Settings".PotZero)
      "Pump_Output"(Disable := "ThrottleDisable", InputValue := "DrillThrottlePotPerFilt", InMin := "Settings".PotZero, InMax := 100.0, OutMin_mA := "Settings".PumpOutMinmA, OutMax_mA := "Settings".PumpOutMaxmA, mAOut => #FlowmAOutTemp)
      wire#w2
      Div(in1 := #FlowmAOutTemp, in2 := 1.0, out => #TDP1RevSetmA)
   END_RUNG
   RUNG wire#w2
      Div(in1 := #FlowmAOutTemp, in2 := 1.0, out => #TDP2RevSetmA)
   END_RUNG
   RUNG wire#w2
      I_Contact( "ThrottleDisable" )
      S_Coil( #TDP1RevEn )
   END_RUNG
   RUNG wire#w2
      I_Contact( "ThrottleDisable" )
      S_Coil( #TDP2RevEn )
   END_RUNG
   RUNG wire#powerrail
      { S7_Templates := "SrcType := Int" } NE_Contact(in1 := #TD_Mode, in2 := #DrillReverse)
      R_Coil( #AllowRev )
   END_RUNG
   // the same network as SCL:
   #_w1 := #TD_Mode = #DrillReverse;
   IF #_w1 AND "TDRotStopped" AND ("DrillThrottlePotPerFilt" <= "Settings".PotZero) THEN
       #AllowRev := TRUE;
   END_IF;
   "Pump_Output"(EN := #_w1 AND #AllowRev AND ("DrillThrottlePotPerFilt" >= "Settings".PotZero),
                 Disable := "ThrottleDisable",
                 InputValue := "DrillThrottlePotPerFilt",
                 InMin := "Settings".PotZero,
                 InMax := 100.0,
                 OutMin_mA := "Settings".PumpOutMinmA,
                 OutMax_mA := "Settings".PumpOutMaxmA,
                 mAOut => #FlowmAOutTemp,
                 ENO => #_w2);
   IF #_w2 THEN
       #TDP1RevSetmA := #FlowmAOutTemp / 1.0;
       #TDP2RevSetmA := #FlowmAOutTemp / 1.0;
   END_IF;
   IF #_w2 AND NOT "ThrottleDisable" THEN
       #TDP1RevEn := TRUE;
       #TDP2RevEn := TRUE;
   END_IF;
   IF #TD_Mode <> #DrillReverse THEN #AllowRev := FALSE; END_IF;
END_REGION

